	(*Valve 13, A+B*)
	(*spare*)
		Valve13FB
			(
			Enable_Motion:= Enable_Motion ,
			Enable_Latch:= TRUE,					(*Enabling Runs Valve as detent type (maintained solenoids*)
			Enable_SideA_PreCharge:= FALSE,		(*Enabling Turns Side A PreCharge Active, reset when Side B is energized in Auto*)
			Enable_SideB_PreCharge:= FALSE,		(*Enabling Turns Side B PreCharge Active, reset when Side A is energized in Auto*)
			PreCharge_Time:= T#0.10S,
			Enable_Auto_Commands:= In_Auto,
			Enable_Manual_Commands:= In_Manual AND All_Robots_Clear,
			In_Manual_SideA_Command:= Discrete_In.ManReqs.24,
			In_Manual_SideB_Command:= Discrete_In.ManReqs.25,
			SideA_Indicator:= FALSE,
			SideB_Indicator:= FALSE,
			TurnOn_SideA_SOL=> N100.Q.24,
			TurnOn_SideB_SOL=> N100.Q.25,
			TurnOn_SideA_Indicator=> Manual_Indicators1.24,
			TurnOn_SideB_Indicator=> Manual_Indicators1.25
			 );
		Valve13FB.In_Auto_SideA_Command:= FALSE;
		Valve13FB.In_Auto_SideB_Command:= FALSE;


	(*Valve 14, A+B*)
	(*spare*)
		Valve14FB
			(
			Enable_Motion:= Enable_Motion ,
			Enable_Latch:= TRUE,					(*Enabling Runs Valve as detent type (maintained solenoids*)
			Enable_SideA_PreCharge:= FALSE,		(*Enabling Turns Side A PreCharge Active, reset when Side B is energized in Auto*)
			Enable_SideB_PreCharge:= FALSE,		(*Enabling Turns Side B PreCharge Active, reset when Side A is energized in Auto*)
			PreCharge_Time:= T#0.10S,
			Enable_Auto_Commands:= In_Auto,
			Enable_Manual_Commands:= In_Manual AND All_Robots_Clear,
			In_Manual_SideA_Command:= Discrete_In.ManReqs.26,
			In_Manual_SideB_Command:= Discrete_In.ManReqs.27,
			SideA_Indicator:= FALSE,
			SideB_Indicator:= FALSE,
			TurnOn_SideA_SOL=> N100.Q.26,
			TurnOn_SideB_SOL=> N100.Q.27,
			TurnOn_SideA_Indicator=> Manual_Indicators1.26,
			TurnOn_SideB_Indicator=> Manual_Indicators1.27
			 );
		Valve14FB.In_Auto_SideA_Command:= FALSE;
		Valve14FB.In_Auto_SideB_Command:= FALSE;


	(*Valve 15, A+B*)
	(*spare*)
		Valve15FB
			(
			Enable_Motion:= Enable_Motion ,
			Enable_Latch:= TRUE,					(*Enabling Runs Valve as detent type (maintained solenoids*)
			Enable_SideA_PreCharge:= FALSE,		(*Enabling Turns Side A PreCharge Active, reset when Side B is energized in Auto*)
			Enable_SideB_PreCharge:= FALSE,		(*Enabling Turns Side B PreCharge Active, reset when Side A is energized in Auto*)
			PreCharge_Time:= T#0.10S,
			Enable_Auto_Commands:= In_Auto,
			Enable_Manual_Commands:= In_Manual AND All_Robots_Clear,
			In_Manual_SideA_Command:= Discrete_In.ManReqs.28,
			In_Manual_SideB_Command:= Discrete_In.ManReqs.29,
			SideA_Indicator:= FALSE,
			SideB_Indicator:= FALSE,
			TurnOn_SideA_SOL=> N100.Q.28,
			TurnOn_SideB_SOL=> N100.Q.29,
			TurnOn_SideA_Indicator=> Manual_Indicators1.28,
			TurnOn_SideB_Indicator=> Manual_Indicators1.29
			 );
		Valve15FB.In_Auto_SideA_Command:= FALSE;
		Valve15FB.In_Auto_SideB_Command:= FALSE;


	(*Valve 16, A+B*)
	(*spare*)
		Valve16FB
			(
			Enable_Motion:= Enable_Motion ,
			Enable_Latch:= TRUE,					(*Enabling Runs Valve as detent type (maintained solenoids*)
			Enable_SideA_PreCharge:= FALSE,		(*Enabling Turns Side A PreCharge Active, reset when Side B is energized in Auto*)
			Enable_SideB_PreCharge:= FALSE,		(*Enabling Turns Side B PreCharge Active, reset when Side A is energized in Auto*)
			PreCharge_Time:= T#0.10S,
			Enable_Auto_Commands:= In_Auto,
			Enable_Manual_Commands:= In_Manual AND All_Robots_Clear,
			In_Manual_SideA_Command:= Discrete_In.ManReqs.30,
			In_Manual_SideB_Command:= Discrete_In.ManReqs.31,
			SideA_Indicator:= FALSE,
			SideB_Indicator:= FALSE,
			TurnOn_SideA_SOL=> N100.Q.30,
			TurnOn_SideB_SOL=> N100.Q.31,
			TurnOn_SideA_Indicator=> Manual_Indicators1.30,
			TurnOn_SideB_Indicator=> Manual_Indicators1.31
			 );
		Valve16FB.In_Auto_SideA_Command:= FALSE;
		Valve16FB.In_Auto_SideB_Command:= FALSE;


























(*end*)
END_ACTION

ACTION ValveBank2:


(*+++++++++++THIS AREA IS CUSTOM PER INSTALLATION AND WILL HAVE TO BE MODIFIED PER +++++++++++++*)
(*+++++++++++THIS AREA IS CUSTOM PER INSTALLATION AND WILL HAVE TO BE MODIFIED PER +++++++++++++*)
(*+++++++++++THIS AREA IS CUSTOM PER INSTALLATION AND WILL HAVE TO BE MODIFIED PER +++++++++++++*)

(*+++++++++++VALVE BANK 2 +++++++++++++*)
(*+++++++++++VALVE BANK 2 +++++++++++++*)
(*+++++++++++VALVE BANK 2 +++++++++++++*)


	(*Valve 17, A+B*)
	(*spare*)
		Valve17FB
			(
			Enable_Motion:= Enable_Motion ,
			Enable_Latch:= TRUE,					(*Enabling Runs Valve as detent type (maintained solenoids*)
			Enable_SideA_PreCharge:= FALSE,		(*Enabling Turns Side A PreCharge Active, reset when Side B is energized in Auto*)
			Enable_SideB_PreCharge:= FALSE,		(*Enabling Turns Side B PreCharge Active, reset when Side A is energized in Auto*)
			PreCharge_Time:= T#0.1S,
			Enable_Auto_Commands:= In_Auto,
			Enable_Manual_Commands:= In_Manual AND All_Robots_Clear,
			In_Manual_SideA_Command:= Discrete_In.ManReqs2.0,
			In_Manual_SideB_Command:= (Discrete_In.ManReqs2.1 OR Discrete_In.Go_Home),
			SideA_Indicator:= FALSE,
			SideB_Indicator:= FALSE,
			TurnOn_SideA_SOL=> N101.Q.0,
			TurnOn_SideB_SOL=> N101.Q.1,
			TurnOn_SideA_Indicator=> Manual_Indicators2.0,
			TurnOn_SideB_Indicator=> Manual_Indicators2.1
			 );
		Valve17FB.In_Auto_SideA_Command:= FALSE;
		Valve17FB.In_Auto_SideB_Command:= FALSE;


	(*Valve 18, A+B*)
	(*spare*)
		Valve18FB
			(
			Enable_Motion:= Enable_Motion ,
			Enable_Latch:= TRUE,					(*Enabling Runs Valve as detent type (maintained solenoids*)
			Enable_SideA_PreCharge:= FALSE,		(*Enabling Turns Side A PreCharge Active, reset when Side B is energized in Auto*)
			Enable_SideB_PreCharge:= FALSE,		(*Enabling Turns Side B PreCharge Active, reset when Side A is energized in Auto*)
			PreCharge_Time:= T#0.10S,
			Enable_Auto_Commands:= In_Auto,
			Enable_Manual_Commands:= In_Manual AND All_Robots_Clear,
			In_Manual_SideA_Command:= Discrete_In.ManReqs2.2,
			In_Manual_SideB_Command:= Discrete_In.ManReqs2.3,
			SideA_Indicator:= FALSE,
			SideB_Indicator:= FALSE,
			TurnOn_SideA_SOL=> N101.Q.2,
			TurnOn_SideB_SOL=> N101.Q.3,
			TurnOn_SideA_Indicator=> Manual_Indicators2.2,
			TurnOn_SideB_Indicator=> Manual_Indicators2.3
			 );
		Valve18FB.In_Auto_SideA_Command:= FALSE;
		Valve18FB.In_Auto_SideB_Command:= FALSE;

	(*Valve 19, A+B*)
	(*spare*)
		Valve19FB
			(
			Enable_Motion:= Enable_Motion ,
			Enable_Latch:= TRUE,					(*Enabling Runs Valve as detent type (maintained solenoids*)
			Enable_SideA_PreCharge:= FALSE,		(*Enabling Turns Side A PreCharge Active, reset when Side B is energized in Auto*)
			Enable_SideB_PreCharge:= FALSE,		(*Enabling Turns Side B PreCharge Active, reset when Side A is energized in Auto*)
			PreCharge_Time:= T#0.10S,
			Enable_Auto_Commands:= In_Auto,
			Enable_Manual_Commands:= In_Manual AND All_Robots_Clear,
			In_Manual_SideA_Command:= Discrete_In.ManReqs2.4,
			In_Manual_SideB_Command:= Discrete_In.ManReqs2.5,
			SideA_Indicator:= FALSE,
			SideB_Indicator:= FALSE,
			TurnOn_SideA_SOL=> N101.Q.4,
			TurnOn_SideB_SOL=> N101.Q.5,
			TurnOn_SideA_Indicator=> Manual_Indicators2.4,
			TurnOn_SideB_Indicator=> Manual_Indicators2.5
			 );
		Valve19FB.In_Auto_SideA_Command:= FALSE;
		Valve19FB.In_Auto_SideB_Command:= FALSE;


	(*Valve 20, A+B*)
	(*spare*)
		Valve20FB
			(
			Enable_Motion:= Enable_Motion ,
			Enable_Latch:= TRUE,					(*Enabling Runs Valve as detent type (maintained solenoids*)
			Enable_SideA_PreCharge:= FALSE,		(*Enabling Turns Side A PreCharge Active, reset when Side B is energized in Auto*)
			Enable_SideB_PreCharge:= FALSE,		(*Enabling Turns Side B PreCharge Active, reset when Side A is energized in Auto*)
			PreCharge_Time:= T#0.10S,
			Enable_Auto_Commands:= In_Auto,
			Enable_Manual_Commands:= In_Manual AND All_Robots_Clear,
			In_Manual_SideA_Command:= Discrete_In.ManReqs2.6,
			In_Manual_SideB_Command:= Discrete_In.ManReqs2.7,
			SideA_Indicator:= FALSE,
			SideB_Indicator:= FALSE,
			TurnOn_SideA_SOL=> N101.Q.6,
			TurnOn_SideB_SOL=> N101.Q.7,
			TurnOn_SideA_Indicator=> Manual_Indicators2.6,
			TurnOn_SideB_Indicator=> Manual_Indicators2.7
			 );
		Valve20FB.In_Auto_SideA_Command:= FALSE;
		Valve20FB.In_Auto_SideB_Command:= FALSE;


	(*Valve 21, A+B*)
	(*spare*)
		Valve21FB
			(
			Enable_Motion:= Enable_Motion ,
			Enable_Latch:= TRUE,					(*Enabling Runs Valve as detent type (maintained solenoids*)
			Enable_SideA_PreCharge:= FALSE,		(*Enabling Turns Side A PreCharge Active, reset when Side B is energized in Auto*)
			Enable_SideB_PreCharge:= FALSE,		(*Enabling Turns Side B PreCharge Active, reset when Side A is energized in Auto*)
			PreCharge_Time:= T#0.10S,
			Enable_Auto_Commands:= In_Auto,
			Enable_Manual_Commands:= In_Manual AND All_Robots_Clear,
			In_Manual_SideA_Command:= Discrete_In.ManReqs2.8,
			In_Manual_SideB_Command:= Discrete_In.ManReqs2.9,
			SideA_Indicator:= FALSE,
			SideB_Indicator:= FALSE,
			TurnOn_SideA_SOL=> N101.Q.8,
			TurnOn_SideB_SOL=> N101.Q.9,
			TurnOn_SideA_Indicator=> Manual_Indicators2.8,
			TurnOn_SideB_Indicator=> Manual_Indicators2.9
			 );
		Valve21FB.In_Auto_SideA_Command:= FALSE;
		Valve21FB.In_Auto_SideB_Command:= FALSE;


	(*Valve 22, A+B*)
	(*spare*)
		Valve22FB
			(
			Enable_Motion:= Enable_Motion ,
			Enable_Latch:= TRUE,					(*Enabling Runs Valve as detent type (maintained solenoids*)
			Enable_SideA_PreCharge:= FALSE,		(*Enabling Turns Side A PreCharge Active, reset when Side B is energized in Auto*)
			Enable_SideB_PreCharge:= FALSE,		(*Enabling Turns Side B PreCharge Active, reset when Side A is energized in Auto*)
			PreCharge_Time:= T#0.10S,
			Enable_Auto_Commands:= In_Auto,
			Enable_Manual_Commands:= In_Manual AND All_Robots_Clear,
			In_Manual_SideA_Command:= Discrete_In.ManReqs2.10,
			In_Manual_SideB_Command:= Discrete_In.ManReqs2.11,
			SideA_Indicator:= FALSE,
			SideB_Indicator:= FALSE,
			TurnOn_SideA_SOL=> N101.Q.10,
			TurnOn_SideB_SOL=> N101.Q.11,
			TurnOn_SideA_Indicator=> Manual_Indicators2.10,
			TurnOn_SideB_Indicator=> Manual_Indicators2.11
			 );
		Valve22FB.In_Auto_SideA_Command:= FALSE;
		Valve22FB.In_Auto_SideB_Command:= FALSE;


	(*Valve 23, A+B*)
	(*spare*)
		Valve23FB
			(
			Enable_Motion:= Enable_Motion ,
			Enable_Latch:= TRUE,					(*Enabling Runs Valve as detent type (maintained solenoids*)
			Enable_SideA_PreCharge:= FALSE,		(*Enabling Turns Side A PreCharge Active, reset when Side B is energized in Auto*)
			Enable_SideB_PreCharge:= FALSE,		(*Enabling Turns Side B PreCharge Active, reset when Side A is energized in Auto*)
			PreCharge_Time:= T#0.10S,
			Enable_Auto_Commands:= In_Auto,
			Enable_Manual_Commands:= In_Manual AND All_Robots_Clear,
			In_Manual_SideA_Command:= Discrete_In.ManReqs2.12,
			In_Manual_SideB_Command:= Discrete_In.ManReqs2.13,
			SideA_Indicator:= FALSE,
			SideB_Indicator:= FALSE,
			TurnOn_SideA_SOL=> N101.Q.12,
			TurnOn_SideB_SOL=> N101.Q.13,
			TurnOn_SideA_Indicator=> Manual_Indicators2.12,
			TurnOn_SideB_Indicator=> Manual_Indicators2.13
			 );
		Valve23FB.In_Auto_SideA_Command:= FALSE;
		Valve23FB.In_Auto_SideB_Command:= FALSE;


	(*Valve 24, A+B*)
	(*spare*)
		Valve24FB
			(
			Enable_Motion:= Enable_Motion ,
			Enable_Latch:= TRUE,					(*Enabling Runs Valve as detent type (maintained solenoids*)
			Enable_SideA_PreCharge:= FALSE,		(*Enabling Turns Side A PreCharge Active, reset when Side B is energized in Auto*)
			Enable_SideB_PreCharge:= FALSE,		(*Enabling Turns Side B PreCharge Active, reset when Side A is energized in Auto*)
			PreCharge_Time:= T#0.10S,
			Enable_Auto_Commands:= In_Auto,
			Enable_Manual_Commands:= In_Manual AND All_Robots_Clear,
			In_Manual_SideA_Command:= Discrete_In.ManReqs2.14,
			In_Manual_SideB_Command:= Discrete_In.ManReqs2.15,
			SideA_Indicator:= FALSE,
			SideB_Indicator:= FALSE,
			TurnOn_SideA_SOL=> N101.Q.14,
			TurnOn_SideB_SOL=> N101.Q.15,
			TurnOn_SideA_Indicator=> Manual_Indicators2.14,
			TurnOn_SideB_Indicator=> Manual_Indicators2.15
			 );
		Valve24FB.In_Auto_SideA_Command:= FALSE;
		Valve24FB.In_Auto_SideB_Command:= FALSE;


	(*Valve 25, A+B*)
	(*spare*)
		Valve25FB
			(
			Enable_Motion:= Enable_Motion ,
			Enable_Latch:= TRUE,					(*Enabling Runs Valve as detent type (maintained solenoids*)
			Enable_SideA_PreCharge:= FALSE,		(*Enabling Turns Side A PreCharge Active, reset when Side B is energized in Auto*)
			Enable_SideB_PreCharge:= FALSE,		(*Enabling Turns Side B PreCharge Active, reset when Side A is energized in Auto*)
			PreCharge_Time:= T#0.10S,
			Enable_Auto_Commands:= In_Auto,
			Enable_Manual_Commands:= In_Manual AND All_Robots_Clear,
			In_Manual_SideA_Command:= Discrete_In.ManReqs2.16,
			In_Manual_SideB_Command:= Discrete_In.ManReqs2.17,
			SideA_Indicator:= FALSE,
			SideB_Indicator:= FALSE,
			TurnOn_SideA_SOL=> N101.Q.16,
			TurnOn_SideB_SOL=> N101.Q.17,
			TurnOn_SideA_Indicator=> Manual_Indicators2.16,
			TurnOn_SideB_Indicator=> Manual_Indicators2.17
			 );
		Valve25FB.In_Auto_SideA_Command:= FALSE;
		Valve25FB.In_Auto_SideB_Command:= FALSE;


	(*Valve 26, A+B*)
	(*spare*)
		Valve26FB
			(
			Enable_Motion:= Enable_Motion ,
			Enable_Latch:= TRUE,					(*Enabling Runs Valve as detent type (maintained solenoids*)
			Enable_SideA_PreCharge:= FALSE,		(*Enabling Turns Side A PreCharge Active, reset when Side B is energized in Auto*)
			Enable_SideB_PreCharge:= FALSE,		(*Enabling Turns Side B PreCharge Active, reset when Side A is energized in Auto*)
			PreCharge_Time:= T#0.10S,
			Enable_Auto_Commands:= In_Auto,
			Enable_Manual_Commands:= In_Manual AND All_Robots_Clear,
			In_Manual_SideA_Command:= Discrete_In.ManReqs2.18,
			In_Manual_SideB_Command:= Discrete_In.ManReqs2.19,
			SideA_Indicator:= FALSE,
			SideB_Indicator:= FALSE,
			TurnOn_SideA_SOL=> N101.Q.18,
			TurnOn_SideB_SOL=> N101.Q.19,
			TurnOn_SideA_Indicator=> Manual_Indicators2.18,
			TurnOn_SideB_Indicator=> Manual_Indicators2.19
			 );
		Valve26FB.In_Auto_SideA_Command:= FALSE;
		Valve26FB.In_Auto_SideB_Command:= FALSE;


	(*Valve 27, A+B*)
	(*spare*)
		Valve27FB
			(
			Enable_Motion:= Enable_Motion ,
			Enable_Latch:= TRUE,					(*Enabling Runs Valve as detent type (maintained solenoids*)
			Enable_SideA_PreCharge:= FALSE,		(*Enabling Turns Side A PreCharge Active, reset when Side B is energized in Auto*)
			Enable_SideB_PreCharge:= FALSE,		(*Enabling Turns Side B PreCharge Active, reset when Side A is energized in Auto*)
			PreCharge_Time:= T#0.10S,
			Enable_Auto_Commands:= In_Auto,
			Enable_Manual_Commands:= In_Manual AND All_Robots_Clear,
			In_Manual_SideA_Command:= Discrete_In.ManReqs2.20,
			In_Manual_SideB_Command:= Discrete_In.ManReqs2.21,
			SideA_Indicator:= FALSE,
			SideB_Indicator:= FALSE,
			TurnOn_SideA_SOL=> N101.Q.20,
			TurnOn_SideB_SOL=> N101.Q.21,
			TurnOn_SideA_Indicator=> Manual_Indicators2.20,
			TurnOn_SideB_Indicator=> Manual_Indicators2.21
			 );
		Valve27FB.In_Auto_SideA_Command:= FALSE;
		Valve27FB.In_Auto_SideB_Command:= FALSE;


	(*Valve 28, A+B*)
	(*spare*)
		Valve28FB
			(
			Enable_Motion:= Enable_Motion ,
			Enable_Latch:= TRUE,					(*Enabling Runs Valve as detent type (maintained solenoids*)
			Enable_SideA_PreCharge:= FALSE,		(*Enabling Turns Side A PreCharge Active, reset when Side B is energized in Auto*)
			Enable_SideB_PreCharge:= FALSE,		(*Enabling Turns Side B PreCharge Active, reset when Side A is energized in Auto*)
			PreCharge_Time:= T#0.10S,
			Enable_Auto_Commands:= In_Auto,
			Enable_Manual_Commands:= In_Manual AND All_Robots_Clear,
			In_Manual_SideA_Command:= Discrete_In.ManReqs2.22,
			In_Manual_SideB_Command:= Discrete_In.ManReqs2.23,
			SideA_Indicator:= FALSE,
			SideB_Indicator:= FALSE,
			TurnOn_SideA_SOL=> N101.Q.22,
			TurnOn_SideB_SOL=> N101.Q.23,
			TurnOn_SideA_Indicator=> Manual_Indicators2.22,
			TurnOn_SideB_Indicator=> Manual_Indicators2.23
			 );
		Valve28FB.In_Auto_SideA_Command:= FALSE;
		Valve28FB.In_Auto_SideB_Command:= FALSE;


	(*Valve 29, A+B*)
	(*spare*)
		Valve29FB
			(
			Enable_Motion:= Enable_Motion ,
			Enable_Latch:= TRUE,					(*Enabling Runs Valve as detent type (maintained solenoids*)
			Enable_SideA_PreCharge:= FALSE,		(*Enabling Turns Side A PreCharge Active, reset when Side B is energized in Auto*)
			Enable_SideB_PreCharge:= FALSE,		(*Enabling Turns Side B PreCharge Active, reset when Side A is energized in Auto*)
			PreCharge_Time:= T#0.10S,
			Enable_Auto_Commands:= In_Auto,
			Enable_Manual_Commands:= In_Manual AND All_Robots_Clear,
			In_Manual_SideA_Command:= Discrete_In.ManReqs2.24,
			In_Manual_SideB_Command:= Discrete_In.ManReqs2.25,
			SideA_Indicator:= FALSE,
			SideB_Indicator:= FALSE,
			TurnOn_SideA_SOL=> N101.Q.24,
			TurnOn_SideB_SOL=> N101.Q.25,
			TurnOn_SideA_Indicator=> Manual_Indicators2.24,
			TurnOn_SideB_Indicator=> Manual_Indicators2.25
			 );
		Valve29FB.In_Auto_SideA_Command:= FALSE;
		Valve29FB.In_Auto_SideB_Command:= FALSE;


	(*Valve 30, A+B*)
	(*spare*)
		Valve30FB
			(
			Enable_Motion:= Enable_Motion ,
			Enable_Latch:= TRUE,					(*Enabling Runs Valve as detent type (maintained solenoids*)
			Enable_SideA_PreCharge:= FALSE,		(*Enabling Turns Side A PreCharge Active, reset when Side B is energized in Auto*)
			Enable_SideB_PreCharge:= FALSE,		(*Enabling Turns Side B PreCharge Active, reset when Side A is energized in Auto*)
			PreCharge_Time:= T#0.10S,
			Enable_Auto_Commands:= In_Auto,
			Enable_Manual_Commands:= In_Manual AND All_Robots_Clear,
			In_Manual_SideA_Command:= Discrete_In.ManReqs2.26,
			In_Manual_SideB_Command:= Discrete_In.ManReqs2.27,
			SideA_Indicator:= FALSE,
			SideB_Indicator:= FALSE,
			TurnOn_SideA_SOL=> N101.Q.26,
			TurnOn_SideB_SOL=> N101.Q.27,
			TurnOn_SideA_Indicator=> Manual_Indicators2.26,
			TurnOn_SideB_Indicator=> Manual_Indicators2.27
			 );
		Valve30FB.In_Auto_SideA_Command:= FALSE;
		Valve30FB.In_Auto_SideB_Command:= FALSE;


	(*Valve 31, A+B*)
	(*spare*)
		Valve31FB
			(
			Enable_Motion:= Enable_Motion ,
			Enable_Latch:= TRUE,					(*Enabling Runs Valve as detent type (maintained solenoids*)
			Enable_SideA_PreCharge:= FALSE,		(*Enabling Turns Side A PreCharge Active, reset when Side B is energized in Auto*)
			Enable_SideB_PreCharge:= FALSE,		(*Enabling Turns Side B PreCharge Active, reset when Side A is energized in Auto*)
			PreCharge_Time:= T#0.10S,
			Enable_Auto_Commands:= In_Auto,
			Enable_Manual_Commands:= In_Manual AND All_Robots_Clear,
			In_Manual_SideA_Command:= Discrete_In.ManReqs2.28,
			In_Manual_SideB_Command:= Discrete_In.ManReqs2.29,
			SideA_Indicator:= FALSE,
			SideB_Indicator:= FALSE,
			TurnOn_SideA_SOL=> N101.Q.28,
			TurnOn_SideB_SOL=> N101.Q.29,
			TurnOn_SideA_Indicator=> Manual_Indicators2.28,
			TurnOn_SideB_Indicator=> Manual_Indicators2.29
			 );
		Valve31FB.In_Auto_SideA_Command:= FALSE;
		Valve31FB.In_Auto_SideB_Command:= FALSE;


	(*Valve 32, A+B*)
	(*spare*)
		Valve32FB
			(
			Enable_Motion:= Enable_Motion ,
			Enable_Latch:= TRUE,					(*Enabling Runs Valve as detent type (maintained solenoids*)
			Enable_SideA_PreCharge:= FALSE,		(*Enabling Turns Side A PreCharge Active, reset when Side B is energized in Auto*)
			Enable_SideB_PreCharge:= FALSE,		(*Enabling Turns Side B PreCharge Active, reset when Side A is energized in Auto*)
			PreCharge_Time:= T#0.10S,
			Enable_Auto_Commands:= In_Auto,
			Enable_Manual_Commands:= In_Manual AND All_Robots_Clear,
			In_Manual_SideA_Command:= Discrete_In.ManReqs2.30,
			In_Manual_SideB_Command:= Discrete_In.ManReqs2.31,
			SideA_Indicator:= FALSE,
			SideB_Indicator:= FALSE,
			TurnOn_SideA_SOL=> N101.Q.30,
			TurnOn_SideB_SOL=> N101.Q.31,
			TurnOn_SideA_Indicator=> Manual_Indicators2.30,
			TurnOn_SideB_Indicator=> Manual_Indicators2.31
			 );
		Valve32FB.In_Auto_SideA_Command:= FALSE;
		Valve32FB.In_Auto_SideB_Command:= FALSE;




















(*end*)
END_ACTION

ACTION ValveBank3:


(*+++++++++++THIS AREA IS CUSTOM PER INSTALLATION AND WILL HAVE TO BE MODIFIED PER +++++++++++++*)
(*+++++++++++THIS AREA IS CUSTOM PER INSTALLATION AND WILL HAVE TO BE MODIFIED PER +++++++++++++*)
(*+++++++++++THIS AREA IS CUSTOM PER INSTALLATION AND WILL HAVE TO BE MODIFIED PER +++++++++++++*)

(*+++++++++++VALVE BANK 3 +++++++++++++*)
(*+++++++++++VALVE BANK 3 +++++++++++++*)
(*+++++++++++VALVE BANK 3 +++++++++++++*)


	(*Valve 33, A+B*)
	(*spare*)
		Valve33FB
			(
			Enable_Motion:= Enable_Motion ,
			Enable_Latch:= TRUE,					(*Enabling Runs Valve as detent type (maintained solenoids*)
			Enable_SideA_PreCharge:= FALSE,		(*Enabling Turns Side A PreCharge Active, reset when Side B is energized in Auto*)
			Enable_SideB_PreCharge:= FALSE,		(*Enabling Turns Side B PreCharge Active, reset when Side A is energized in Auto*)
			PreCharge_Time:= T#0.1S,
			Enable_Auto_Commands:= In_Auto,
			Enable_Manual_Commands:= In_Manual AND All_Robots_Clear,
			In_Manual_SideA_Command:= Discrete_In.ManReqs3.0,
			In_Manual_SideB_Command:= (Discrete_In.ManReqs3.1 OR Discrete_In.Go_Home),
			SideA_Indicator:= FALSE,
			SideB_Indicator:= FALSE,
			TurnOn_SideA_SOL=> N102.Q.0,
			TurnOn_SideB_SOL=> N102.Q.1,
			TurnOn_SideA_Indicator=> Manual_Indicators3.0,
			TurnOn_SideB_Indicator=> Manual_Indicators3.1
			 );
		Valve33FB.In_Auto_SideA_Command:= FALSE;
		Valve33FB.In_Auto_SideB_Command:= FALSE;


	(*Valve 34, A+B*)
	(*spare*)
		Valve34FB
			(
			Enable_Motion:= Enable_Motion ,
			Enable_Latch:= TRUE,					(*Enabling Runs Valve as detent type (maintained solenoids*)
			Enable_SideA_PreCharge:= FALSE,		(*Enabling Turns Side A PreCharge Active, reset when Side B is energized in Auto*)
			Enable_SideB_PreCharge:= FALSE,		(*Enabling Turns Side B PreCharge Active, reset when Side A is energized in Auto*)
			PreCharge_Time:= T#0.10S,
			Enable_Auto_Commands:= In_Auto,
			Enable_Manual_Commands:= In_Manual AND All_Robots_Clear,
			In_Manual_SideA_Command:= Discrete_In.ManReqs3.2,
			In_Manual_SideB_Command:= Discrete_In.ManReqs3.3,
			SideA_Indicator:= FALSE,
			SideB_Indicator:= FALSE,
			TurnOn_SideA_SOL=> N102.Q.2,
			TurnOn_SideB_SOL=> N102.Q.3,
			TurnOn_SideA_Indicator=> Manual_Indicators3.2,
			TurnOn_SideB_Indicator=> Manual_Indicators3.3
			 );
		Valve34FB.In_Auto_SideA_Command:= FALSE;
		Valve34FB.In_Auto_SideB_Command:= FALSE;


	(*Valve 35, A+B*)
	(*spare*)
		Valve35FB
			(
			Enable_Motion:= Enable_Motion ,
			Enable_Latch:= TRUE,					(*Enabling Runs Valve as detent type (maintained solenoids*)
			Enable_SideA_PreCharge:= FALSE,		(*Enabling Turns Side A PreCharge Active, reset when Side B is energized in Auto*)
			Enable_SideB_PreCharge:= FALSE,		(*Enabling Turns Side B PreCharge Active, reset when Side A is energized in Auto*)
			PreCharge_Time:= T#0.10S,
			Enable_Auto_Commands:= In_Auto,
			Enable_Manual_Commands:= In_Manual AND All_Robots_Clear,
			In_Manual_SideA_Command:= Discrete_In.ManReqs3.4,
			In_Manual_SideB_Command:= Discrete_In.ManReqs3.5,
			SideA_Indicator:= FALSE,
			SideB_Indicator:= FALSE,
			TurnOn_SideA_SOL=> N102.Q.4,
			TurnOn_SideB_SOL=> N102.Q.5,
			TurnOn_SideA_Indicator=> Manual_Indicators3.4,
			TurnOn_SideB_Indicator=> Manual_Indicators3.5
			 );
		Valve35FB.In_Auto_SideA_Command:= FALSE;
		Valve35FB.In_Auto_SideB_Command:= FALSE;


	(*Valve 36, A+B*)
	(*spare*)
		Valve36FB
			(
			Enable_Motion:= Enable_Motion ,
			Enable_Latch:= TRUE,					(*Enabling Runs Valve as detent type (maintained solenoids*)
			Enable_SideA_PreCharge:= FALSE,		(*Enabling Turns Side A PreCharge Active, reset when Side B is energized in Auto*)
			Enable_SideB_PreCharge:= FALSE,		(*Enabling Turns Side B PreCharge Active, reset when Side A is energized in Auto*)
			PreCharge_Time:= T#0.10S,
			Enable_Auto_Commands:= In_Auto,
			Enable_Manual_Commands:= In_Manual AND All_Robots_Clear,
			In_Manual_SideA_Command:= Discrete_In.ManReqs3.6,
			In_Manual_SideB_Command:= Discrete_In.ManReqs3.7,
			SideA_Indicator:= FALSE,
			SideB_Indicator:= FALSE,
			TurnOn_SideA_SOL=> N102.Q.6,
			TurnOn_SideB_SOL=> N102.Q.7,
			TurnOn_SideA_Indicator=> Manual_Indicators3.6,
			TurnOn_SideB_Indicator=> Manual_Indicators3.7
			 );
		Valve36FB.In_Auto_SideA_Command:= FALSE;
		Valve36FB.In_Auto_SideB_Command:= FALSE;


	(*Valve 37, A+B*)
	(*spare*)
		Valve37FB
			(
			Enable_Motion:= Enable_Motion ,
			Enable_Latch:= TRUE,					(*Enabling Runs Valve as detent type (maintained solenoids*)
			Enable_SideA_PreCharge:= FALSE,		(*Enabling Turns Side A PreCharge Active, reset when Side B is energized in Auto*)
			Enable_SideB_PreCharge:= FALSE,		(*Enabling Turns Side B PreCharge Active, reset when Side A is energized in Auto*)
			PreCharge_Time:= T#0.10S,
			Enable_Auto_Commands:= In_Auto,
			Enable_Manual_Commands:= In_Manual AND All_Robots_Clear,
			In_Manual_SideA_Command:= Discrete_In.ManReqs3.8,
			In_Manual_SideB_Command:= Discrete_In.ManReqs3.9,
			SideA_Indicator:= FALSE,
			SideB_Indicator:= FALSE,
			TurnOn_SideA_SOL=> N102.Q.8,
			TurnOn_SideB_SOL=> N102.Q.9,
			TurnOn_SideA_Indicator=> Manual_Indicators3.8,
			TurnOn_SideB_Indicator=> Manual_Indicators3.9
			 );
		Valve37FB.In_Auto_SideA_Command:= FALSE;
		Valve37FB.In_Auto_SideB_Command:= FALSE;


	(*Valve 38, A+B*)
	(*spare*)
		Valve38FB
			(
			Enable_Motion:= Enable_Motion ,
			Enable_Latch:= TRUE,					(*Enabling Runs Valve as detent type (maintained solenoids*)
			Enable_SideA_PreCharge:= FALSE,		(*Enabling Turns Side A PreCharge Active, reset when Side B is energized in Auto*)
			Enable_SideB_PreCharge:= FALSE,		(*Enabling Turns Side B PreCharge Active, reset when Side A is energized in Auto*)
			PreCharge_Time:= T#0.10S,
			Enable_Auto_Commands:= In_Auto,
			Enable_Manual_Commands:= In_Manual AND All_Robots_Clear,
			In_Manual_SideA_Command:= Discrete_In.ManReqs3.10,
			In_Manual_SideB_Command:= Discrete_In.ManReqs3.11,
			SideA_Indicator:= FALSE,
			SideB_Indicator:= FALSE,
			TurnOn_SideA_SOL=> N102.Q.10,
			TurnOn_SideB_SOL=> N102.Q.11,
			TurnOn_SideA_Indicator=> Manual_Indicators3.10,
			TurnOn_SideB_Indicator=> Manual_Indicators3.11
			 );
		Valve38FB.In_Auto_SideA_Command:= FALSE;
		Valve38FB.In_Auto_SideB_Command:= FALSE;


	(*Valve 39, A+B*)
	(*spare*)
		Valve39FB
			(
			Enable_Motion:= Enable_Motion ,
			Enable_Latch:= TRUE,					(*Enabling Runs Valve as detent type (maintained solenoids*)
			Enable_SideA_PreCharge:= FALSE,		(*Enabling Turns Side A PreCharge Active, reset when Side B is energized in Auto*)
			Enable_SideB_PreCharge:= FALSE,		(*Enabling Turns Side B PreCharge Active, reset when Side A is energized in Auto*)
			PreCharge_Time:= T#0.10S,
			Enable_Auto_Commands:= In_Auto,
			Enable_Manual_Commands:= In_Manual AND All_Robots_Clear,
			In_Manual_SideA_Command:= Discrete_In.ManReqs3.12,
			In_Manual_SideB_Command:= Discrete_In.ManReqs3.13,
			SideA_Indicator:= FALSE,
			SideB_Indicator:= FALSE,
			TurnOn_SideA_SOL=> N102.Q.12,
			TurnOn_SideB_SOL=> N102.Q.13,
			TurnOn_SideA_Indicator=> Manual_Indicators3.12,
			TurnOn_SideB_Indicator=> Manual_Indicators3.13
			 );
		Valve39FB.In_Auto_SideA_Command:= FALSE;
		Valve39FB.In_Auto_SideB_Command:= FALSE;


	(*Valve 40, A+B*)
	(*spare*)
		Valve40FB
			(
			Enable_Motion:= Enable_Motion ,
			Enable_Latch:= TRUE,					(*Enabling Runs Valve as detent type (maintained solenoids*)
			Enable_SideA_PreCharge:= FALSE,		(*Enabling Turns Side A PreCharge Active, reset when Side B is energized in Auto*)
			Enable_SideB_PreCharge:= FALSE,		(*Enabling Turns Side B PreCharge Active, reset when Side A is energized in Auto*)
			PreCharge_Time:= T#0.10S,
			Enable_Auto_Commands:= In_Auto,
			Enable_Manual_Commands:= In_Manual AND All_Robots_Clear,
			In_Manual_SideA_Command:= Discrete_In.ManReqs3.14,
			In_Manual_SideB_Command:= Discrete_In.ManReqs3.15,
			SideA_Indicator:= FALSE,
			SideB_Indicator:= FALSE,
			TurnOn_SideA_SOL=> N102.Q.14,
			TurnOn_SideB_SOL=> N102.Q.15,
			TurnOn_SideA_Indicator=> Manual_Indicators3.14,
			TurnOn_SideB_Indicator=> Manual_Indicators3.15
			 );
		Valve40FB.In_Auto_SideA_Command:= FALSE;
		Valve40FB.In_Auto_SideB_Command:= FALSE;


	(*Valve 41, A+B*)
	(*spare*)
		Valve41FB
			(
			Enable_Motion:= Enable_Motion ,
			Enable_Latch:= TRUE,					(*Enabling Runs Valve as detent type (maintained solenoids*)
			Enable_SideA_PreCharge:= FALSE,		(*Enabling Turns Side A PreCharge Active, reset when Side B is energized in Auto*)
			Enable_SideB_PreCharge:= FALSE,		(*Enabling Turns Side B PreCharge Active, reset when Side A is energized in Auto*)
			PreCharge_Time:= T#0.10S,
			Enable_Auto_Commands:= In_Auto,
			Enable_Manual_Commands:= In_Manual AND All_Robots_Clear,
			In_Manual_SideA_Command:= Discrete_In.ManReqs3.16,
			In_Manual_SideB_Command:= Discrete_In.ManReqs3.17,
			SideA_Indicator:= FALSE,
			SideB_Indicator:= FALSE,
			TurnOn_SideA_SOL=> N102.Q.16,
			TurnOn_SideB_SOL=> N102.Q.17,
			TurnOn_SideA_Indicator=> Manual_Indicators3.16,
			TurnOn_SideB_Indicator=> Manual_Indicators3.17
			 );
		Valve41FB.In_Auto_SideA_Command:= FALSE;
		Valve41FB.In_Auto_SideB_Command:= FALSE;


	(*Valve 42, A+B*)
	(*spare*)
		Valve42FB
			(
			Enable_Motion:= Enable_Motion ,
			Enable_Latch:= TRUE,					(*Enabling Runs Valve as detent type (maintained solenoids*)
			Enable_SideA_PreCharge:= FALSE,		(*Enabling Turns Side A PreCharge Active, reset when Side B is energized in Auto*)
			Enable_SideB_PreCharge:= FALSE,		(*Enabling Turns Side B PreCharge Active, reset when Side A is energized in Auto*)
			PreCharge_Time:= T#0.10S,
			Enable_Auto_Commands:= In_Auto,
			Enable_Manual_Commands:= In_Manual AND All_Robots_Clear,
			In_Manual_SideA_Command:= Discrete_In.ManReqs3.18,
			In_Manual_SideB_Command:= Discrete_In.ManReqs3.19,
			SideA_Indicator:= FALSE,
			SideB_Indicator:= FALSE,
			TurnOn_SideA_SOL=> N102.Q.18,
			TurnOn_SideB_SOL=> N102.Q.19,
			TurnOn_SideA_Indicator=> Manual_Indicators3.18,
			TurnOn_SideB_Indicator=> Manual_Indicators3.19
			 );
		Valve42FB.In_Auto_SideA_Command:= FALSE;
		Valve42FB.In_Auto_SideB_Command:= FALSE;


	(*Valve 43, A+B*)
	(*spare*)
		Valve43FB
			(
			Enable_Motion:= Enable_Motion ,
			Enable_Latch:= TRUE,					(*Enabling Runs Valve as detent type (maintained solenoids*)
			Enable_SideA_PreCharge:= FALSE,		(*Enabling Turns Side A PreCharge Active, reset when Side B is energized in Auto*)
			Enable_SideB_PreCharge:= FALSE,		(*Enabling Turns Side B PreCharge Active, reset when Side A is energized in Auto*)
			PreCharge_Time:= T#0.10S,
			Enable_Auto_Commands:= In_Auto,
			Enable_Manual_Commands:= In_Manual AND All_Robots_Clear,
			In_Manual_SideA_Command:= Discrete_In.ManReqs3.20,
			In_Manual_SideB_Command:= Discrete_In.ManReqs3.21,
			SideA_Indicator:= FALSE,
			SideB_Indicator:= FALSE,
			TurnOn_SideA_SOL=> N102.Q.20,
			TurnOn_SideB_SOL=> N102.Q.21,
			TurnOn_SideA_Indicator=> Manual_Indicators3.20,
			TurnOn_SideB_Indicator=> Manual_Indicators3.21
			 );
		Valve43FB.In_Auto_SideA_Command:= FALSE;
		Valve43FB.In_Auto_SideB_Command:= FALSE;


	(*Valve 44, A+B*)
	(*spare*)
		Valve44FB
			(
			Enable_Motion:= Enable_Motion ,
			Enable_Latch:= TRUE,					(*Enabling Runs Valve as detent type (maintained solenoids*)
			Enable_SideA_PreCharge:= FALSE,		(*Enabling Turns Side A PreCharge Active, reset when Side B is energized in Auto*)
			Enable_SideB_PreCharge:= FALSE,		(*Enabling Turns Side B PreCharge Active, reset when Side A is energized in Auto*)
			PreCharge_Time:= T#0.10S,
			Enable_Auto_Commands:= In_Auto,
			Enable_Manual_Commands:= In_Manual AND All_Robots_Clear,
			In_Manual_SideA_Command:= Discrete_In.ManReqs3.22,
			In_Manual_SideB_Command:= Discrete_In.ManReqs3.23,
			SideA_Indicator:= FALSE,
			SideB_Indicator:= FALSE,
			TurnOn_SideA_SOL=> N102.Q.22,
			TurnOn_SideB_SOL=> N102.Q.23,
			TurnOn_SideA_Indicator=> Manual_Indicators3.22,
			TurnOn_SideB_Indicator=> Manual_Indicators3.23
			 );
		Valve44FB.In_Auto_SideA_Command:= FALSE;
		Valve44FB.In_Auto_SideB_Command:= FALSE;


	(*Valve 45, A+B*)
	(*spare*)
		Valve45FB
			(
			Enable_Motion:= Enable_Motion ,
			Enable_Latch:= TRUE,					(*Enabling Runs Valve as detent type (maintained solenoids*)
			Enable_SideA_PreCharge:= FALSE,		(*Enabling Turns Side A PreCharge Active, reset when Side B is energized in Auto*)
			Enable_SideB_PreCharge:= FALSE,		(*Enabling Turns Side B PreCharge Active, reset when Side A is energized in Auto*)
			PreCharge_Time:= T#0.10S,
			Enable_Auto_Commands:= In_Auto,
			Enable_Manual_Commands:= In_Manual AND All_Robots_Clear,
			In_Manual_SideA_Command:= Discrete_In.ManReqs3.24,
			In_Manual_SideB_Command:= Discrete_In.ManReqs3.25,
			SideA_Indicator:= FALSE,
			SideB_Indicator:= FALSE,
			TurnOn_SideA_SOL=> N102.Q.24,
			TurnOn_SideB_SOL=> N102.Q.25,
			TurnOn_SideA_Indicator=> Manual_Indicators3.24,
			TurnOn_SideB_Indicator=> Manual_Indicators3.25
			 );
		Valve45FB.In_Auto_SideA_Command:= FALSE;
		Valve45FB.In_Auto_SideB_Command:= FALSE;


	(*Valve 46, A+B*)
	(*spare*)
		Valve46FB
			(
			Enable_Motion:= Enable_Motion ,
			Enable_Latch:= TRUE,					(*Enabling Runs Valve as detent type (maintained solenoids*)
			Enable_SideA_PreCharge:= FALSE,		(*Enabling Turns Side A PreCharge Active, reset when Side B is energized in Auto*)
			Enable_SideB_PreCharge:= FALSE,		(*Enabling Turns Side B PreCharge Active, reset when Side A is energized in Auto*)
			PreCharge_Time:= T#0.10S,
			Enable_Auto_Commands:= In_Auto,
			Enable_Manual_Commands:= In_Manual AND All_Robots_Clear,
			In_Manual_SideA_Command:= Discrete_In.ManReqs3.26,
			In_Manual_SideB_Command:= Discrete_In.ManReqs3.27,
			SideA_Indicator:= FALSE,
			SideB_Indicator:= FALSE,
			TurnOn_SideA_SOL=> N102.Q.26,
			TurnOn_SideB_SOL=> N102.Q.27,
			TurnOn_SideA_Indicator=> Manual_Indicators3.26,
			TurnOn_SideB_Indicator=> Manual_Indicators3.27
			 );
		Valve46FB.In_Auto_SideA_Command:= FALSE;
		Valve46FB.In_Auto_SideB_Command:= FALSE;


	(*Valve 47, A+B*)
	(*spare*)
		Valve47FB
			(
			Enable_Motion:= Enable_Motion ,
			Enable_Latch:= TRUE,					(*Enabling Runs Valve as detent type (maintained solenoids*)
			Enable_SideA_PreCharge:= FALSE,		(*Enabling Turns Side A PreCharge Active, reset when Side B is energized in Auto*)
			Enable_SideB_PreCharge:= FALSE,		(*Enabling Turns Side B PreCharge Active, reset when Side A is energized in Auto*)
			PreCharge_Time:= T#0.10S,
			Enable_Auto_Commands:= In_Auto,
			Enable_Manual_Commands:= In_Manual AND All_Robots_Clear,
			In_Manual_SideA_Command:= Discrete_In.ManReqs3.28,
			In_Manual_SideB_Command:= Discrete_In.ManReqs3.29,
			SideA_Indicator:= FALSE,
			SideB_Indicator:= FALSE,
			TurnOn_SideA_SOL=> N102.Q.28,
			TurnOn_SideB_SOL=> N102.Q.29,
			TurnOn_SideA_Indicator=> Manual_Indicators3.28,
			TurnOn_SideB_Indicator=> Manual_Indicators3.29
			 );
		Valve47FB.In_Auto_SideA_Command:= FALSE;
		Valve47FB.In_Auto_SideB_Command:= FALSE;


	(*Valve 48, A+B*)
	(*spare*)
		Valve48FB
			(
			Enable_Motion:= Enable_Motion ,
			Enable_Latch:= TRUE,					(*Enabling Runs Valve as detent type (maintained solenoids*)
			Enable_SideA_PreCharge:= FALSE,		(*Enabling Turns Side A PreCharge Active, reset when Side B is energized in Auto*)
			Enable_SideB_PreCharge:= FALSE,		(*Enabling Turns Side B PreCharge Active, reset when Side A is energized in Auto*)
			PreCharge_Time:= T#0.10S,
			Enable_Auto_Commands:= In_Auto,
			Enable_Manual_Commands:= In_Manual AND All_Robots_Clear,
			In_Manual_SideA_Command:= Discrete_In.ManReqs3.30,
			In_Manual_SideB_Command:= Discrete_In.ManReqs3.31,
			SideA_Indicator:= FALSE,
			SideB_Indicator:= FALSE,
			TurnOn_SideA_SOL=> N102.Q.30,
			TurnOn_SideB_SOL=> N102.Q.31,
			TurnOn_SideA_Indicator=> Manual_Indicators3.30,
			TurnOn_SideB_Indicator=> Manual_Indicators3.31
			 );
		Valve48FB.In_Auto_SideA_Command:= FALSE;
		Valve48FB.In_Auto_SideB_Command:= FALSE;


























(*end*)
END_ACTION

ACTION Xfer_To_UI:
(*Transfer General Status of Fixture and I/O Images for Display On HMI*)
	Discrete_Image.Status:= Status;
	Discrete_Image.CLFaults1:= CLFaults1;
	Discrete_Image.CLFaults2:= CLFaults2;
	Discrete_Image.CLFaults3:= CLFaults3;
	Discrete_Image.CLFaults4:= CLFaults4;
	Discrete_Image.CLFaulted:= CLFaulted;
	Discrete_Image.PPFaults:= PPFaults;
	Discrete_Image.PPFaults1:= PPFaults1;
	Discrete_Image.PPFaults2:= PPFaults2;
	Discrete_Image.PPFaulted:= PPFaulted;
	Discrete_Image.Model_Data:= Model_ID;
	Discrete_Image.ToolID:= Fix_ID;
	Discrete_Image.ProdCount:= Prod_Count_Out;
	Discrete_Image.CycleTime:= Cycle_Time_Out;
	Discrete_Image.PrevCycleTime:= PrevCycle_Time_Out;
	Discrete_Image.LoadTime:= Load_Time_Out;
	Discrete_Image.WeldTime:= Weld_Time_Out;
	Discrete_Image.UnloadTime:= Unload_Time_Out;

	Discrete_Image.InAuto:= In_Auto_Mode;
	Discrete_Image.InManual:= In_Manual_Mode;
	Discrete_Image.ManInds:= Manual_Indicators1;
	Discrete_Image.ManInds2:= Manual_Indicators2;
	Discrete_Image.ManInds3:= Manual_Indicators3;
	Discrete_Image.At_Home:= Tool_At_Home;
	Discrete_Image.Enable_Motion:= Enable_Motion;
	Discrete_Image.All_Sensors_Off:= All_Sensors_Off;
	Discrete_Image.Bypass_ACKS:= Discrete_In.Bypass_REQS;
	Discrete_Image.CustomApplication_ACKS:= Discrete_In.CustomApplication_REQS;
	Discrete_Image.Fixture_Allow_Model_Change:= Fixture_Allow_Model_Change;
	Discrete_Image.NodeLayout:=NodeLayout;
	Discrete_Image.NodeState:=NodeState;
	
	Discrete_Image.Input_Node_Count:= Discrete_In.Input_Node_Count;
	Discrete_Image.VB_Node_Count:= Discrete_In.VB_Node_Count;
	Discrete_Image.Water_Stand_Count:= Discrete_In.Water_Stand_Count;

	IF  (Discrete_Image.Input_Node_Count < 4)
		THEN Discrete_Image.VB_Screen_Position:= 1;
	ELSIF  (Discrete_Image.Input_Node_Count < 7)
		THEN Discrete_Image.VB_Screen_Position:= 2;
	ELSIF  (Discrete_Image.Input_Node_Count < 10)
		THEN Discrete_Image.VB_Screen_Position:= 3;
	ELSIF  (Discrete_Image.Input_Node_Count < 13)
		THEN Discrete_Image.VB_Screen_Position:= 4;
	ELSIF  (Discrete_Image.Input_Node_Count < 16)
		THEN Discrete_Image.VB_Screen_Position:= 5;
	ELSIF  (Discrete_Image.Input_Node_Count < 19)
		THEN Discrete_Image.VB_Screen_Position:= 6;
	ELSIF  (Discrete_Image.Input_Node_Count < 22)
		THEN Discrete_Image.VB_Screen_Position:= 7;
	ELSIF  (Discrete_Image.Input_Node_Count < 26)
		THEN Discrete_Image.VB_Screen_Position:= 8;
	ELSE
			Discrete_Image.VB_Screen_Position:= 9;
	END_IF;

	Discrete_Image.N00:= N00;
	Discrete_Image.N01:= N01;
	Discrete_Image.N02:= N02;
	Discrete_Image.N03:= N03;
	Discrete_Image.N04:= N04;
	Discrete_Image.N05:= N05;
	Discrete_Image.N06:= N06;
	Discrete_Image.N07:= N07;
	Discrete_Image.N08:= N08;
	Discrete_Image.N09:= N09;
	Discrete_Image.N10:= N10;
	Discrete_Image.N11:= N11;
	Discrete_Image.N12:= N12;
	Discrete_Image.N13:= N13;
	Discrete_Image.N14:= N14;
	Discrete_Image.N15:= N15;
	Discrete_Image.N16:= N16;
	Discrete_Image.N17:= N17;
	Discrete_Image.N18:= N18;
	Discrete_Image.N19:= N19;
	Discrete_Image.N100:= N100;
	Discrete_Image.N100_STAT:= N100_STAT;
	Discrete_Image.N101:= N101;
	Discrete_Image.N101_STAT:= N101_STAT;
	Discrete_Image.N102:= N102;
	Discrete_Image.N102_STAT:= N102_STAT;


	Discrete_Image.ECatSlave_Cable_Breaks:= ECatSlave_Cable_Breaks;

	Discrete_Image.Operator_Performance_Pen:= Production_Report.Shift_Report[0].Prod_Performance;
END_ACTION

END_PROGRAM

// ---- POUs/Fixtures and EOAT/Not_Used/Fix11.TcPOU
(*Fixture*)

PROGRAM Fix11
	VAR_INPUT
		Enable_Prog: BOOL;
		Enable_Motion: BOOL;
		Discrete_In: udt_FixXX_Input_Image_20180202;
		Dry_Cycle: BOOL;
		Cell_In_Services: BOOL;
		Flash_Rate: BOOL;
		NodeLayout:udt_ECATNodeData_20221507;

	END_VAR

	VAR
(*Hardware Related Data Types*)
			(*Develop "Beckhoff Nodes"*)
			{attribute 'OPC.UA.DA':='1'}
			N00 AT %I*: udt_EP1111;
			{attribute 'OPC.UA.DA':='1'}
			N01 AT %I*: udt_EP1008_002_v2;
			{attribute 'OPC.UA.DA':='1'}
			N02 AT %I*: udt_EP1008_002_v2;
			{attribute 'OPC.UA.DA':='1'}
			N03 AT %I*: udt_EP1008_002_v2;
			{attribute 'OPC.UA.DA':='1'}
			N04 AT %I*: udt_EP1008_002_v2;
			{attribute 'OPC.UA.DA':='1'}
			N05 AT %I*: udt_EP1008_002_v2;
			{attribute 'OPC.UA.DA':='1'}
			N06 AT %I*: udt_EP1008_002_v2;
			{attribute 'OPC.UA.DA':='1'}
			N07 AT %I*: udt_EP1008_002_v2;
			{attribute 'OPC.UA.DA':='1'}
			N08 AT %I*: udt_EP1008_002_v2;
			{attribute 'OPC.UA.DA':='1'}
			N09 AT %I*: udt_EP1008_002_v2;
			{attribute 'OPC.UA.DA':='1'}
			N10 AT %I*: udt_EP1008_002_v2;
			{attribute 'OPC.UA.DA':='1'}
			N11 AT %I*: udt_EP1008_002_v2;
			{attribute 'OPC.UA.DA':='1'}
			N12 AT %I*: udt_EP1008_002_v2;
			{attribute 'OPC.UA.DA':='1'}
			N13 AT %I*: udt_EP1008_002_v2;
			{attribute 'OPC.UA.DA':='1'}
			N14 AT %I*: udt_EP1008_002_v2;
			{attribute 'OPC.UA.DA':='1'}
			N15 AT %I*: udt_EP1008_002_v2;
			{attribute 'OPC.UA.DA':='1'}
			N16 AT %I*: udt_EP1008_002_v2;
			{attribute 'OPC.UA.DA':='1'}
			N17 AT %I*: udt_EP1008_002_v2;
			{attribute 'OPC.UA.DA':='1'}
			N18 AT %I*: udt_EP1008_002_v2;
			{attribute 'OPC.UA.DA':='1'}
			N19 AT %I*: udt_EP1008_002_v2;
			{attribute 'OPC.UA.DA':='1'}
			N20 AT %I*: udt_EP1008_002_v2;
			{attribute 'OPC.UA.DA':='1'}
			N21 AT %I*: udt_EP1008_002_v2;
			{attribute 'OPC.UA.DA':='1'}
			N22 AT %I*: udt_EP1008_002_v2;
			{attribute 'OPC.UA.DA':='1'}
			N100 AT %Q*: udt_SMC_EX260_ValveBank;
			{attribute 'OPC.UA.DA':='1'}
			N100_STAT AT %I*:udt_SMC_EX260_Stat;
			{attribute 'OPC.UA.DA':='1'}
			N101 AT %Q*: udt_SMC_EX260_ValveBank;
			{attribute 'OPC.UA.DA':='1'}
			N101_STAT AT %I*:udt_SMC_EX260_Stat;
			{attribute 'OPC.UA.DA':='1'}
			N102 AT %Q*: udt_SMC_EX260_ValveBank;
			{attribute 'OPC.UA.DA':='1'}
			N102_STAT AT %I*:udt_SMC_EX260_Stat;

(* Nodes States*)
		NodeState: ARRAY[0..63] OF UINT;
		DiscreteNode_OK: BOOL;
(*Cable Break States*)
		ECatSlave_Cable_Breaks: ARRAY[0..1] OF DINT;
(*Standard Internal Variables*)
		(*Generic Sensor Variables*)
		All_Sensors_On: UINT;
		All_Sensors_Off: BOOL;
		All_Sensors_Off1: BOOL;
		All_Sensors_Off2: BOOL;
		(*Generic Position Variables*)
		Tool_At_Home: BOOL;
		Tool_At_Load: UINT;
		Tool_At_Weld: UINT;
		Tool_At_Rotate: UINT;
		Tool_At_Seal: UINT;
		Tool_At_Stud: UINT;
		Tool_At_Unload: UINT ;
		(*Grouping Of Items*)
		All_QAChecks_OK: BOOL;
		QAChecks_Failed: BOOL;
		(*General Internals*)
		In_Auto: BOOL;
		In_Manual: BOOL;

		Auto_Run: BOOL;
		Reset_All_Completes:BOOL;
		Load_Robots_Clear1: BOOL;
		Load_Robots_Clear2: BOOL;
		Load_Robots_Clear: BOOL;
		Load_Robots_WorkingOK1: BOOL;
		Load_Robots_WorkingOK2: BOOL;
		Load_Robots_Complete1: BOOL;
		Load_Robots_Complete2: BOOL;
		Load_Robots_PartInEOAT1: BOOL;
		Load_Robots_PartInEOAT2: BOOL;
		Load_Robots_UnclampEarly1: BOOL;
		Load_Robots_UnclampEarly2: BOOL;
		Seal_Robots_Clear: BOOL;
		Seal_Robots_WorkingOK: BOOL;
		Seal_Robots_UnclampEarly: BOOL;
		Seal_Robots_Complete: BOOL;
		Stud_Robots_Clear: BOOL;
		Stud_Robots_WorkingOK: BOOL;
		Stud_Robots_UnclampEarly: BOOL;
		Stud_Robots_Complete: BOOL;
		Weld_Robots_Clear: BOOL;
		Weld_Robots_WorkingOK: BOOL;
		Weld_Robots_UnclampEarly: BOOL;
		Weld_Robots_Complete: BOOL;
		Mig_Robots_Ready :BOOL;
		TurntableA_Clear: BOOL;
		TurntableB_Clear: BOOL;
		Turntable_Clear:BOOL;
		Turntable_WorkingOK: BOOL;
		TurntableA_Complete: BOOL;
		TurntableB_Complete: BOOL;
		Unload_Robots_Clear1: BOOL;
		Unload_Robots_WorkingOK1: BOOL;
		Unload_Robots_Complete1: BOOL;
		Unload_Robots_EOATEmpty1: BOOL;
		Unload_Robots_Clear2: BOOL;
		Unload_Robots_WorkingOK2: BOOL;
		Unload_Robots_Complete2: BOOL;
		Unload_Robots_EOATEmpty2: BOOL;
		Unload_Robots_Clear: BOOL;
		All_Robots_Clear: BOOL;

		Unload_Robot_Complete: BOOL;

		Start_Load_Robots1: BOOL;
		Start_Load_Robots2: BOOL;
		Start_Weld_Robots: BOOL;
		Start_Unload_Robots1: BOOL;
		Start_Unload_Robots2: BOOL;
		Start_Seal_Robots: BOOL;
		Start_Stud_Robots: BOOL;
		Start_TurntableA: BOOL;
		Start_TurntableB: BOOL;
		Load_Robots_Proceed1: BOOL;
		Load_Robots_Proceed2: BOOL;
		Weld_Robots_Proceed: BOOL;
		Seal_Robots_Proceed: BOOL;
		Stud_Robots_Proceed: BOOL;
		Unload_Robots_Proceed1: BOOL;
		Unload_Robots_Proceed2: BOOL;

		Prod_Inc: R_TRIG;
		Cycle_Time: TON;
		Cycle_Time_Pulse: R_TRIG;
		Load_Time: TON;
		Weld_Time: TON;
		Seal_Time: TON;
		Stud_Time: TON;
		Turn_Time: TON;
		Unload_Time: TON;
		Date_Stamp_TMR: TON;
		Date_StampHome_TMR: TON;
		CLFaulted: UDINT;
		PPFaulted: UDINT;
		Manual_Ind_HomePrompt: BOOL;
		Fixture_Allow_Model_Change: BOOL;

(*Non-Standard Variables*)

		(*FB Instances*)
		Clamp1FB: FB_Cylinder_Status;
		Clamp2FB: FB_Cylinder_Status;
		Clamp3FB: FB_Cylinder_Status;
		Clamp4FB: FB_Cylinder_Status;
		Clamp5FB: FB_Cylinder_Status;
		Clamp6FB: FB_Cylinder_Status;
		Clamp7FB: FB_Cylinder_Status;
		Clamp8FB: FB_Cylinder_Status;
		Clamp9FB: FB_Cylinder_Status;
		Clamp10FB: FB_Cylinder_Status;
		Clamp11FB: FB_Cylinder_Status;
		Clamp12FB: FB_Cylinder_Status;
		Clamp13FB: FB_Cylinder_Status;
		Clamp14FB: FB_Cylinder_Status;
		Clamp15FB: FB_Cylinder_Status;
		Clamp16FB: FB_Cylinder_Status;
		Clamp17FB: FB_Cylinder_Status;
		Clamp18FB: FB_Cylinder_Status;
		Clamp19FB: FB_Cylinder_Status;
		Clamp20FB: FB_Cylinder_Status;
		Clamp21FB: FB_Cylinder_Status;
		Clamp22FB: FB_Cylinder_Status;
		Clamp23FB: FB_Cylinder_Status;
		Clamp24FB: FB_Cylinder_Status;
		Cyl1FB: FB_TripleCylinder_20150625;
		Pin1FB: FB_Cylinder_Status;
		Pin2FB: FB_Cylinder_Status;
		Pin3FB: FB_Cylinder_Status;
		Pin4FB: FB_Cylinder_Status;
		Pin5FB: FB_Cylinder_Status;
		Pin6FB: FB_Cylinder_Status;
		Pin7FB: FB_Cylinder_Status;
		Pin8FB: FB_Cylinder_Status;
		Pin9FB: FB_Cylinder_Status;
		Pin10FB: FB_Cylinder_Status;
		Pin11FB: FB_Cylinder_Status;
		Pin12FB: FB_Cylinder_Status;
		Pin13FB: FB_Cylinder_Status;
		Pin14FB: FB_Cylinder_Status;
		Slide1FB: FB_Cylinder_Status;
		Slide2FB: FB_Cylinder_Status;
		Slide3FB: FB_Cylinder_Status;
		Slide4FB: FB_Cylinder_Status;
		Slide5FB: FB_Cylinder_Status;
		Slide6FB: FB_Cylinder_Status;
		Swing1FB: FB_Cylinder_Status;
		Swing2FB: FB_Cylinder_Status;
		Swing3FB: FB_Cylinder_Status;
		Swing4FB: FB_Cylinder_Status;
		Swing5FB: FB_Cylinder_Status;
		Swing6FB: FB_Cylinder_Status;
		QACheck1FB: FB_Cylinder_Status;
		QACheck2FB: FB_Cylinder_Status;
		CheckQA1FB: FB_GTAC_QAcheck_20150529;
		Part_Present1FB: FB_PP_Sensor;
		Part_Present2FB: FB_PP_Sensor;
		Part_Present3FB: FB_PP_Sensor;
		Part_Present4FB: FB_PP_Sensor;
		Part_Present5FB: FB_PP_Sensor;
		Part_Present6FB: FB_PP_Sensor;
		Part_Present7FB: FB_PP_Sensor;
		Part_Present8FB: FB_PP_Sensor;
		Part_Present9FB: FB_PP_Sensor;
		Part_Present10FB: FB_PP_Sensor;
		Part_Present11FB: FB_PP_Sensor;
		Part_Present12FB: FB_PP_Sensor;
		Part_Present13FB: FB_PP_Sensor;
		Part_Present14FB: FB_PP_Sensor;
		Part_Present15FB: FB_PP_Sensor;
		Part_Present16FB: FB_PP_Sensor;
		Part_Present17FB: FB_PP_Sensor;
		Part_Present18FB: FB_PP_Sensor;
		Part_Present19FB: FB_PP_Sensor;
		Part_Present20FB: FB_PP_Sensor;
		Part_Present21FB: FB_PP_Sensor;
		Part_Present22FB: FB_PP_Sensor;
		Part_Present23FB: FB_PP_Sensor;
		Part_Present24FB: FB_PP_Sensor;
		Part_Present25FB: FB_PP_Sensor;
		Part_Present26FB: FB_PP_Sensor;
		Part_Present27FB: FB_PP_Sensor;
		Part_Present28FB: FB_PP_Sensor;
		Part_Present29FB: FB_PP_Sensor;
		Part_Present30FB: FB_PP_Sensor;
		Part_Present31FB: FB_PP_Sensor;
		Part_Present32FB: FB_PP_Sensor;
		Part_Present33FB: FB_PP_Sensor;
		Part_Present34FB: FB_PP_Sensor;
		Part_Present35FB: FB_PP_Sensor;
		Part_Present36FB: FB_PP_Sensor;
		Part_Present37FB: FB_PP_Sensor;
		Part_Present38FB: FB_PP_Sensor;
		Part_Present39FB: FB_PP_Sensor;
		Part_Present40FB: FB_PP_Sensor;
		Tape_Present1FB: FB_PP_Sensor;

		(*Valve FBs*)
		Valve1FB: FB_GTAC_Valve_20170704;
		Valve2FB: FB_GTAC_Valve_20170704;
		Valve3FB: FB_GTAC_Valve_20170704;
		Valve4FB: FB_GTAC_Valve_20170704;
		Valve5FB: FB_GTAC_Valve_20170704;
		Valve6FB: FB_GTAC_Valve_20170704;
		Valve7FB: FB_GTAC_Valve_20170704;
		Valve8FB: FB_GTAC_Valve_20170704;
		Valve9FB: FB_GTAC_Valve_20170704;
		Valve10FB: FB_GTAC_Valve_20170704;
		Valve11FB: FB_GTAC_Valve_20170704;
		Valve12FB: FB_GTAC_Valve_20170704;
		Valve13FB: FB_GTAC_Valve_20170704;
		Valve14FB: FB_GTAC_Valve_20170704;
		Valve15FB: FB_GTAC_Valve_20170704;
		Valve16FB: FB_GTAC_Valve_20170704;
		Valve17FB: FB_GTAC_Valve_20170704;
		Valve18FB: FB_GTAC_Valve_20170704;
		Valve19FB: FB_GTAC_Valve_20170704;
		Valve20FB: FB_GTAC_Valve_20170704;
		Valve21FB: FB_GTAC_Valve_20170704;
		Valve22FB: FB_GTAC_Valve_20170704;
		Valve23FB: FB_GTAC_Valve_20170704;
		Valve24FB: FB_GTAC_Valve_20170704;
		Valve25FB: FB_GTAC_Valve_20170704;
		Valve26FB: FB_GTAC_Valve_20170704;
		Valve27FB: FB_GTAC_Valve_20170704;
		Valve28FB: FB_GTAC_Valve_20170704;
		Valve29FB: FB_GTAC_Valve_20170704;
		Valve30FB: FB_GTAC_Valve_20170704;
		Valve31FB: FB_GTAC_Valve_20170704;
		Valve32FB: FB_GTAC_Valve_20170704;
		Valve33FB: FB_GTAC_Valve_20170704;
		Valve34FB: FB_GTAC_Valve_20170704;
		Valve35FB: FB_GTAC_Valve_20170704;
		Valve36FB: FB_GTAC_Valve_20170704;
		Valve37FB: FB_GTAC_Valve_20170704;
		Valve38FB: FB_GTAC_Valve_20170704;
		Valve39FB: FB_GTAC_Valve_20170704;
		Valve40FB: FB_GTAC_Valve_20170704;
		Valve41FB: FB_GTAC_Valve_20170704;
		Valve42FB: FB_GTAC_Valve_20170704;
		Valve43FB: FB_GTAC_Valve_20170704;
		Valve44FB: FB_GTAC_Valve_20170704;
		Valve45FB: FB_GTAC_Valve_20170704;
		Valve46FB: FB_GTAC_Valve_20170704;
		Valve47FB: FB_GTAC_Valve_20170704;
		Valve48FB: FB_GTAC_Valve_20170704;

		(*Tool Positions*)
			(*Add User Indivdual Position Variables Here*)
			Clamp1ADVD: BOOL;
			Clamp1RETD: BOOL;
			Clamp2ADVD: BOOL;
			Clamp2RETD: BOOL;
			Clamp3ADVD: BOOL;
			Clamp3RETD: BOOL;
			Clamp4ADVD: BOOL;
			Clamp4RETD: BOOL;
			Clamp5ADVD: BOOL;
			Clamp5RETD: BOOL;
			Clamp6ADVD: BOOL;
			Clamp6RETD: BOOL;
			Clamp7ADVD: BOOL;
			Clamp7RETD: BOOL;
			Clamp8ADVD: BOOL;
			Clamp8RETD: BOOL;
			Clamp9ADVD: BOOL;
			Clamp9RETD: BOOL;
			Clamp10ADVD: BOOL;
			Clamp10RETD: BOOL;
			Clamp11ADVD: BOOL;
			Clamp11RETD: BOOL;
			Clamp12ADVD: BOOL;
			Clamp12RETD: BOOL;
			Clamp13ADVD: BOOL;
			Clamp13RETD: BOOL;
			Clamp14ADVD: BOOL;
			Clamp14RETD: BOOL;
			Clamp15ADVD: BOOL;
			Clamp15RETD: BOOL;
			Clamp16ADVD: BOOL;
			Clamp16RETD: BOOL;
			Clamp17ADVD: BOOL;
			Clamp17RETD: BOOL;
			Clamp18ADVD: BOOL;
			Clamp18RETD: BOOL;
			Clamp19ADVD: BOOL;
			Clamp19RETD: BOOL;
			Clamp20ADVD: BOOL;
			Clamp20RETD: BOOL;
			Clamp21ADVD: BOOL;
			Clamp21RETD: BOOL;
			Clamp22ADVD: BOOL;
			Clamp22RETD: BOOL;
			Clamp23ADVD: BOOL;
			Clamp23RETD: BOOL;
			Clamp24ADVD: BOOL;
			Clamp24RETD: BOOL;
			Cyl1ADVD: BOOL;
			Cyl1MID: BOOL;
			Cyl1RETD: BOOL;
			Pin1ADVD: BOOL;
			Pin1RETD: BOOL;
			Pin2ADVD: BOOL;
			Pin2RETD: BOOL;
			Pin3ADVD: BOOL;
			Pin3RETD: BOOL;
			Pin4ADVD: BOOL;
			Pin4RETD: BOOL;
			Pin5ADVD: BOOL;
			Pin5RETD: BOOL;
			Pin6ADVD: BOOL;
			Pin6RETD: BOOL;
			Pin7ADVD: BOOL;
			Pin7RETD: BOOL;
			Pin8ADVD: BOOL;
			Pin8RETD: BOOL;
			Pin9ADVD: BOOL;
			Pin9RETD: BOOL;
			Pin10ADVD: BOOL;
			Pin10RETD: BOOL;
			Pin11ADVD: BOOL;
			Pin11RETD: BOOL;
			Pin12ADVD: BOOL;
			Pin12RETD: BOOL;
			Pin13ADVD: BOOL;
			Pin13RETD: BOOL;
			Pin14ADVD: BOOL;
			Pin14RETD: BOOL;
			Slide1ADVD: BOOL;
			Slide1RETD: BOOL;
			Slide2ADVD: BOOL;
			Slide2RETD: BOOL;
			Slide3ADVD: BOOL;
			Slide3RETD: BOOL;
			Slide4ADVD: BOOL;
			Slide4RETD: BOOL;
			Slide5ADVD: BOOL;
			Slide5RETD: BOOL;
			Slide6ADVD: BOOL;
			Slide6RETD: BOOL;
			Swing1ADVD: BOOL;
			Swing1RETD: BOOL;
			Swing2ADVD: BOOL;
			Swing2RETD: BOOL;
			Swing3ADVD: BOOL;
			Swing3RETD: BOOL;
			Swing4ADVD: BOOL;
			Swing4RETD: BOOL;
			Swing5ADVD: BOOL;
			Swing5RETD: BOOL;
			Swing6ADVD: BOOL;
			Swing6RETD: BOOL;
			QACheck1ADVD: BOOL;
			QACheck1RETD: BOOL;
			QACheck2ADVD: BOOL;
			QACheck2RETD: BOOL;

		(*Part Present Sensors*)
			(*Main Body Present*)
			Part_Present1: BOOL;
			Part_Present2: BOOL;
			Part_Present3: BOOL;
			Part_Present4: BOOL;
			Part_Present5: BOOL;
			Part_Present6: BOOL;
			Part_Present7: BOOL;
			Part_Present8: BOOL;
			Part_Present9: BOOL;
			Part_Present10: BOOL;
			Part_Present11: BOOL;
			Part_Present12: BOOL;
			Part_Present13: BOOL;
			Part_Present14: BOOL;
			Part_Present15: BOOL;
			Part_Present16: BOOL;
			Part_Present17: BOOL;
			Part_Present18: BOOL;
			Part_Present19: BOOL;
			Part_Present20: BOOL;
			Part_Present21: BOOL;
			Part_Present22: BOOL;
			Part_Present23: BOOL;
			Part_Present24: BOOL;
			Part_Present25: BOOL;
			Part_Present26: BOOL;
			Part_Present27: BOOL;
			Part_Present28: BOOL;
			Part_Present29: BOOL;
			Part_Present30: BOOL;
			Part_Present31: BOOL;
			Part_Present32: BOOL;
			Part_Present33: BOOL;
			Part_Present34: BOOL;
			Part_Present35: BOOL;
			Part_Present36: BOOL;
			Part_Present37: BOOL;
			Part_Present38: BOOL;
			Part_Present39: BOOL;
			Part_Present40: BOOL;
			Tape_Present1: BOOL;

		(*Motion Sequence Variables*)
			Clamp_Step: UINT;
			Repo1_Step: UINT;
			Repo2_Step: UINT;
			Repo3_Step: UINT;
			Repo4_Step: UINT;
			Unclamp_Step: UINT;

		(*Custom Application Variables*)
			Weld_Curtain_Bypass: BOOL;
			Vacuum_Bypass: BOOL;
			Sealer_Bypass: BOOL;
			Stud_Bypass: BOOL;
			Turntable_Bypassed: BOOL;
			Door_Open: BOOL;

END_VAR

	(*data that needs to be retained in the event of a power cycle*)
	VAR PERSISTENT

		Load_Complete1: BOOL;
		Load_Complete2: BOOL;
		Load_Complete: BOOL;
		Stud_Complete: BOOL;
		Welding_Complete: BOOL;
		Sealing_Complete: BOOL;
		Unload_Complete: BOOL;
		TurnA_Complete: BOOL;
		TurnB_Complete: BOOL;
		Cycle_Complete: BOOL;
		Eject_Complete: BOOL;
		VacCheck_Complete: BOOL;
		Date_Stamp_Complete: BOOL;
		Load_Seq01: FB_GTAC_Load_Seq_20230302;
		Production_Count:INT;
		Repo_REQS: UINT;
		(*Allow_Load_PreCall: BOOL;
		Allow_Weld_PreCall: BOOL;
		Allow_Unload_PreCall: BOOL;*)
		(*All_SubPP_Off: BOOL;*)
		Production_Report: FB_Production_Report_20221007;

	END_VAR

	VAR_OUTPUT

		Prog_Ok: BOOL;
		Discrete_Image: udt_FixXX_Output_Image_20220715;
		In_Auto_Mode: BOOL;
		In_Manual_Mode: BOOL;
		Manual_Indicators1: DINT;
		Manual_Indicators2: DINT;
		Manual_Indicators3: DINT;
		At_Home: BOOL;
		Ready_To_Load: BOOL;
		Red_Lamp_Req: BOOL;
		Status: UINT;
		CLFaults1:UDINT;
		CLFaults2:UDINT;
		CLFaults3:UDINT;
		CLFaults4:UDINT;
		PPFaults: UDINT;
		PPFaults1: UDINT;
		PPFaults2: UDINT;
		Prod_Count_Out: INT;
		Cycle_Time_Out: TIME;
		PrevCycle_Time_Out: TIME;
		Load_Time_Out: TIME;
		Weld_Time_Out: TIME;
		Seal_Time_Out: TIME;
		Stud_Time_Out: TIME;
		Turn_Time_Out: TIME;
		Unload_Time_Out: TIME;
		Model_ID: UINT;
		TurntableA_At_Robot: BOOL;
		TurntableB_At_Robot: BOOL;
		Tool_Call_ForLoadRobots1: BOOL;
		Tool_Call_ForLoadRobots2: BOOL;
		Tool_Call_ForSealRobots: BOOL;
		Tool_Call_ForStudRobots: BOOL;
		Tool_Call_ForWeldRobots: BOOL;
		Tool_Call_ForSweepA: BOOL;
		Tool_Call_ForSweepB: BOOL;
		Tool_Call_ForUnloadRobots1: BOOL;
		Tool_Call_ForUnloadRobots2: BOOL;
		Robots_Clear_ToProceed: BOOL;
		Task_ID: UINT;
		Fix_ID: UINT;
		Load_Complete1_Ack: BOOL;
		Load_Complete2_Ack: BOOL;
		Seal_Complete_Ack: BOOL;
		Stud_Complete_Ack: BOOL;
		Weld_Complete_Ack: BOOL;
		TurnA_Complete_Ack: BOOL;
		TurnB_Complete_Ack: BOOL;
		Unload_Complete1_Ack: BOOL;
		Unload_Complete2_Ack: BOOL;
		Repo_Ack: UINT;
		Door_Close_Req: BOOL;
		Door_Open_Req: BOOL;
	END_VAR

	(*Set FB_OK to True*)
	Prog_OK:= TRUE;


	(*Set conditions to allow model change*)
	Fixture_Allow_Model_Change:= (In_Manual AND Tool_At_Home AND All_Sensors_Off AND All_Robots_Clear)
							OR (Model_ID=0);



(*$$$$$$$$$$$$$$$$$$$$$$$$$$$$$$$$$$$$$$$$$$$$ Fixture Bypasses $$$$$$$$$$$$$$$$$$$$$$$$$$$$$$$$$$$$$$$$$$$$$$$$$$$$*)
	Weld_Curtain_Bypass:= Discrete_In.Bypass_REQS.0;
	Vacuum_Bypass:= Discrete_In.Bypass_REQS.1;
	Stud_Bypass:= Discrete_In.Bypass_REQS.2;
	Turntable_Bypassed:= ((TurntableA_At_Robot AND Tool_At_Home AND All_Sensors_OFF)
					OR (Turntable_Bypassed AND NOT TurntableB_At_Robot))
					OR Discrete_In.Bypass_REQS.3;
	Sealer_Bypass:= MAIN.SL01.Disp1_Bypass;


(*$$$$$$$$$$$$$$$$$$$$$$$$$$$$$$$$$$$$$$$$$$$$ Gather Status Of Hardware $$$$$$$$$$$$$$$$$$$$$$$$$$$$$$$$$$$$$$$$$$$$$$$$$$$$*)
	(*Check on Status of Hardware*)
	Hardware();

(*$$$$$$$$$$$$$$$$$$$$$$$$$$$$$$$$$$$$$$$$$$$$$ Gather Standard Inputs $$$$$$$$$$$$$$$$$$$$$$$$$$$$$$$$$$$$$$$$$$$$$$$$$$$$$$$$$*)

(*Clamp/Cylinder Inputs*)
	Cylinders();

(*Part Present Inputs*)
	Proxies();

(*$$$$$$$$$$$$$$$$$$$$$$$$$$$$$$$$$$$$$$$$$$$ Qaulity Checking Routines $$$$$$$$$$$$$$$$$$$$$$$$$$$$$$$$$$$$$$$$$$$$$$$$$$$$$$$$$*)

	(*QA Checks*)
		CheckQA1FB(
			Start_QAcheck:= Auto_Run AND Enable_Motion AND Tool_At_Load.3,
			QAcheck_Reset:= Cycle_Complete OR (In_Manual AND Discrete_In.Go_Home AND All_Sensors_Off),
			QAcheck_Retry:= In_From_ICxx.QA_Reset.0,
			QAcheck_Release:= In_From_ICxx.QA_Reset.1,
			QAcheck_Adv_In:= QACheck1ADVD AND QACheck2ADVD,
			QAcheck_Ret_In:= QACheck1RETD AND QACheck2RETD,
			User_Dry_Cycle:= Dry_Cycle,
			QAcheck_OK_Delay:= T#0.75s,
			QAcheck_Fault_Delay:= T#3.0s,
			QAcheck_OK=> All_QAChecks_OK,
			QAcheck_Failed=> QAChecks_Failed);



(*$$$$$$$$$$$$$$$$$$$$$$$$$$$$$$$$$$$$$$$$$$$$$$$$ Internal Code $$$$$$$$$$$$$$$$$$$$$$$$$$$$$$$$$$$$$$$$$$$$$$$$$$$$$$$$$$$$$$$$$$$$*)
(*Auto / Manual Mode Code*)
	IF Discrete_In.Mode_Select.0 AND NOT Discrete_In.Mode_Select.1
		THEN
			In_Auto:= TRUE;
			In_Auto_Mode:= TRUE;
	END_IF;
	IF NOT Discrete_In.Mode_Select.0 AND Discrete_In.Mode_Select.1
		THEN
			In_Auto:= FALSE;
			In_Auto_Mode:= FALSE;
	END_IF;
	In_Manual:= NOT In_Auto;
	In_Manual_Mode:= In_Manual;

(*--------------------------------------------------------------------------------Tool Positions---------------------------------------------------------------*)
	Tool_States();

(*----------------------------------------------------Part Present Sensor Input Patterns----------------------------------------------------------------*)
	All_Sensors();


(*>>>>>>>>>>>>>>>>>>>>>>>>>>>>>>>>>>>>>>>>>> Auto Run Cycle >>>>>>>>>>>>>>>>>>>>>>>>>>>>>>>>>>>>>>>*)
(*+++++++++++THIS AREA IS CUSTOM PER INSTALLATION AND WILL HAVE TO BE MODIFIED PER +++++++++++++*)
(*+++++++++++THIS AREA IS CUSTOM PER INSTALLATION AND WILL HAVE TO BE MODIFIED PER +++++++++++++*)
	(*Control of Auto_Run*)
	Auto_Run:= Enable_Motion AND In_Auto AND Model_ID<>0 AND NOT Cycle_Complete;

	(*Auto Run Enables All Other Auto Cycle Code*)
	IF Auto_Run
		THEN

			IF (NOT Load_Complete1 OR (Load_Robots_UnclampEarly1 AND All_Sensors_On.1))
				AND Load_Robots_Clear2 AND Stud_Robots_Clear AND Seal_Robots_Clear
				AND Weld_Robots_Clear AND TurnTable_Clear AND Unload_Robots_Clear
				AND TurnTableA_At_Robot
				THEN
					(*Start 1st Load Robots*)
					Start_Load_Robots1:= ((Tool_At_Load.0 AND All_Sensors_Off AND NOT Repo_Reqs.0 AND Load_Robots_PartInEOAT1)
									OR (Tool_At_Load.1 AND All_Sensors_On.4 AND Repo_Reqs.0))
									OR Load_Robots_WorkingOK1;
					(*Allow 1st Load Robots To Proceed*)
					Load_Robots_Proceed1:= Tool_At_Load.0 AND All_Sensors_Off AND Load_Robots_PartInEOAT1;
			ELSE
					Start_Load_Robots1:= FALSE;
					Load_Robots_Proceed1:= FALSE;
			END_IF;


			IF (NOT Load_Complete2 OR (Load_Robots_UnclampEarly2 AND All_Sensors_On.2))
				AND Load_Robots_Clear1 AND Stud_Robots_Clear AND Seal_Robots_Clear
				AND Weld_Robots_Clear AND TurnTable_Clear AND Unload_Robots_Clear
				AND TurnTableA_At_Robot
				THEN
					(*Start 2nd Load Robots*)
					Start_Load_Robots2:= ((Tool_At_Load.1 AND All_Sensors_Off AND NOT Repo_Reqs.0 AND Load_Robots_PartInEOAT2)
									OR (Tool_At_Load.1 AND All_Sensors_On.4 AND Repo_Reqs.0))
									OR Load_Robots_WorkingOK2;
					(*Allow 2nd Load Robots To Proceed*)
					Load_Robots_Proceed2:= Tool_At_Load.1 AND All_Sensors_Off AND Load_Robots_PartInEOAT2;
			ELSE
					Start_Load_Robots2:= FALSE;
					Load_Robots_Proceed2:= FALSE;
			END_IF;


			IF NOT Sealer_Bypass AND Load_Complete AND NOT Sealing_Complete
				AND Load_Robots_Clear AND Stud_Robots_Clear AND  Weld_Robots_Clear AND TurnTable_Clear AND Unload_Robots_Clear
				AND TurnTableA_At_Robot
				THEN
					(*Start Seal Robots*)
					Start_Seal_Robots:= ((Tool_At_Seal.0 AND All_Sensors_On.3 AND NOT Repo_Reqs.1 AND NOT MAIN.SL01.Disp1_Faulted AND MAIN.SL01.Disp1_Ready)
									OR (Tool_At_Seal.1 AND All_Sensors_On.4 AND Repo_Reqs.1))
									OR Seal_Robots_WorkingOK;
					(*Allow Seal Robots To Proceed*)
					Seal_Robots_Proceed:= Tool_At_Seal.0 AND All_Sensors_On.3;
			ELSE
					Start_Seal_Robots:= FALSE;
					Seal_Robots_Proceed:= FALSE;
			END_IF;


			IF NOT Stud_Bypass AND Load_Complete AND NOT Stud_Complete AND NOT Welding_Complete
				AND Load_Robots_Clear AND Seal_Robots_Clear AND  Weld_Robots_Clear AND TurnTable_Clear AND Unload_Robots_Clear
				AND TurnTableA_At_Robot
				THEN
					(*Start Stud Robots*)
					Start_Stud_Robots:= ((Tool_At_Stud.0 AND All_Sensors_On.3 AND NOT Repo_Reqs.2)
									OR (Tool_At_Stud.1 AND All_Sensors_On.4 AND Repo_Reqs.2))
									OR Stud_Robots_WorkingOK;
					(*Allow Stud Robots To Proceed*)
					Stud_Robots_Proceed:= Tool_At_Stud.0 AND All_Sensors_On.3;
			ELSE
					Start_Stud_Robots:= FALSE;
					Stud_Robots_Proceed:= FALSE;
			END_IF;


                             IF  NOT TurnA_Complete AND Load_Complete AND NOT Welding_Complete AND NOT Unload_Complete
				 AND Load_Robots_Clear AND Seal_Robots_Clear AND Stud_Robots_Clear AND  Weld_Robots_Clear AND Unload_Robots_Clear
				AND (NOT TurntableA_At_Robot OR TurnTable_WorkingOK)
				THEN
					(*Start Turntable SweepA (Fix01 to the Robot)*)
					Start_TurntableA:= ((Tool_At_Rotate.0 AND All_Sensors_On.3)
									OR (All_Sensors_Off AND Tool_At_Home))
									OR TurnTable_WorkingOK;
			ELSE
					Start_TurntableA:= FALSE;
			END_IF;


			IF NOT TurnB_Complete AND Welding_Complete AND NOT Unload_Complete AND (Sealing_Complete OR Sealer_Bypass) AND (Stud_Complete OR Stud_Bypass)
				AND Load_Robots_Clear AND Seal_Robots_Clear AND Stud_Robots_Clear AND Weld_Robots_Clear  AND Unload_Robots_Clear
				AND (NOT TurntableB_At_Robot OR TurnTable_WorkingOK)
				THEN
					(*Start Turntable SweepB (Fix01 to the Operator)*)
					Start_TurntableB:= TRUE;
                             ELSIF All_Sensors_Off AND NOT TurnB_Complete AND Weld_Robots_Clear AND Load_Robots_Clear AND Unload_Robots_Clear
				AND (NOT TurntableB_At_Robot OR TurnTable_WorkingOK)
			THEN
					Start_TurntableB:= All_Sensors_Off;
                             ELSE
					Start_TurntableB:= FALSE;
                             END_IF;


			IF Load_Complete AND NOT Welding_Complete AND (Sealing_Complete OR Sealer_Bypass) AND (Stud_Complete OR Stud_Bypass) AND NOT Unload_Complete
				AND Load_Robots_Clear AND Seal_Robots_Clear AND Stud_Robots_Clear AND TurnTable_Clear AND Unload_Robots_Clear
				AND TurnTableA_At_Robot AND Mig_Robots_Ready 
				THEN
					(*Start Weld Robots*)
					Start_Weld_Robots:=((Tool_At_Weld.0 AND NOT Repo_Reqs.3 AND NOT Repo_Reqs.4 AND NOT Repo_Reqs.5 AND All_Sensors_On.3)
										OR (Tool_At_Weld.1 AND Repo_Reqs.3 AND All_Sensors_On.3)
										OR (Tool_At_Weld.2 AND Repo_Reqs.4 AND All_Sensors_On.4)
										OR (Tool_At_Weld.3 AND Repo_Reqs.5 AND All_Sensors_On.5)
										OR (Tool_At_Unload.0 AND Weld_Robots_UnclampEarly))
										OR Weld_Robots_WorkingOK;
					(*Allow Weld Robots To Proceed*)
					Weld_Robots_Proceed:= Load_Complete AND Tool_At_Weld.0 AND All_Sensors_On.3;
			ELSE
					Start_Weld_Robots:= FALSE;
					Weld_Robots_Proceed:= FALSE;
			END_IF;


			IF Welding_Complete  AND (Sealing_Complete OR Sealer_Bypass) AND (Stud_Complete OR Stud_Bypass) AND NOT Unload_Complete
				AND Load_Robots_Clear AND Seal_Robots_Clear AND Stud_Robots_Clear AND TurnTable_Clear AND Unload_Robots_Clear2
				AND TurnTableA_At_Robot
				THEN
					(*Start Unload Robots*)
					Start_Unload_Robots1:=((((Tool_At_Unload.0 AND NOT Repo_Reqs.6 AND NOT Repo_Reqs.7 AND All_Sensors_On.8)
										OR (Tool_At_Unload.1 AND Repo_Reqs.6)
										OR (Tool_At_Unload.2 AND Repo_Reqs.7))
										AND (All_Sensors_On.8 AND Unload_Robots_EOATEmpty1))
										OR (NOT Unload_Robots_Clear1 AND NOT Unload_Robots_EOATEmpty1))
										OR Unload_Robots_WorkingOK1;
					(*Allow Unload Robots To Proceed*)
					Unload_Robots_Proceed1:= Welding_Complete AND Tool_At_Unload.0 AND All_Sensors_On.8 AND Unload_Robots_EOATEmpty1;
			ELSE
					Start_Unload_Robots1:= FALSE;
					Unload_Robots_Proceed1:= FALSE;
			END_IF;


			IF Welding_Complete  AND (Sealing_Complete OR Sealer_Bypass) AND (Stud_Complete OR Stud_Bypass) AND NOT Unload_Complete
				AND Load_Robots_Clear AND Seal_Robots_Clear AND Stud_Robots_Clear AND TurnTable_Clear AND Unload_Robots_Clear1
				AND TurnTableA_At_Robot
				THEN
					(*Start Unload Robots*)
					Start_Unload_Robots2:=((((Tool_At_Unload.0 AND NOT Repo_Reqs.6 AND NOT Repo_Reqs.7 AND All_Sensors_On.8)
										OR (Tool_At_Unload.1 AND Repo_Reqs.6)
										OR (Tool_At_Unload.2 AND Repo_Reqs.7))
										AND (All_Sensors_On.8 AND Unload_Robots_EOATEmpty2))
										OR (NOT Unload_Robots_Clear2 AND NOT Unload_Robots_EOATEmpty2))
										OR Unload_Robots_WorkingOK2;
					(*Allow Unload Robots To Proceed*)
					Unload_Robots_Proceed2:= Welding_Complete AND Tool_At_Unload.0 AND All_Sensors_On.8 AND Unload_Robots_EOATEmpty2;
			ELSE
					Start_Unload_Robots2:= FALSE;
					Unload_Robots_Proceed2:= FALSE;
			END_IF;


	ELSE
		Start_Load_Robots1:= FALSE;
		Start_Load_Robots2:= FALSE;
		Start_Seal_Robots:= FALSE;
		Start_Stud_Robots:= FALSE;
		Start_TurntableA:= FALSE;
		Start_TurntableB:= FALSE;
		Start_Weld_Robots:= FALSE;
		Start_Unload_Robots1:= FALSE;
		Start_Unload_Robots2:= FALSE;
		Load_Robots_Proceed1:=FALSE;
		Load_Robots_Proceed2:=FALSE;
		Seal_Robots_Proceed:=FALSE;
		Weld_Robots_Proceed:=FALSE;
		Unload_Robots_Proceed1:=FALSE;
		Unload_Robots_Proceed2:=FALSE;
	END_IF;




(*---------------------------------------------------------------Completes----------------------------------------------------*)
	(*1st Load Complete*)
	IF NOT Dry_Cycle
		THEN
		Load_Complete1:=  All_Sensors_On.1;
	ELSIF Dry_Cycle
		THEN
		IF Tool_At_Home AND Enable_Motion AND All_Sensors_Off
			THEN
			Load_Complete1:= TRUE;
		END_IF;
	END_IF;
	(*2nd Load Complete*)
	IF NOT Dry_Cycle
		THEN
		Load_Complete2:=  All_Sensors_On.2;
	ELSIF Dry_Cycle
		THEN
		IF Tool_At_Home AND Enable_Motion AND All_Sensors_Off
			THEN
			Load_Complete2:= TRUE;
		END_IF;
	END_IF;
	(*All Load Complete*)
	IF NOT Dry_Cycle
		THEN
		Load_Complete:= (All_Sensors_On.2
					OR (All_Sensors_On.3 AND Tool_At_Weld.0)
					OR (Repo_Reqs.0 AND All_Sensors_On.4)
					OR (Repo_Reqs.1 AND All_Sensors_On.5)
					OR (Repo_Reqs.2 AND All_Sensors_On.6))
					OR Weld_Robots_WorkingOK OR Welding_Complete;
	ELSIF Dry_Cycle
		THEN
		IF Load_Complete1 AND Load_Complete2 AND All_Sensors_Off
			THEN
			Load_Complete:= TRUE;
		END_IF;
	END_IF;

	(*Welding Complete*)
	IF Weld_Robots_Complete
		THEN
		Welding_Complete:= TRUE;
	END_IF;

	(*Unload Complete*)
	IF NOT Dry_Cycle
		THEN
			IF (Unload_Robots_Complete1 OR Unload_Robots_Complete2 OR (All_Sensors_Off AND Unload_Robots_Clear)) AND Welding_Complete
				THEN
				Unload_Complete:= TRUE;
			END_IF;
	ELSIF Dry_Cycle
		THEN
			IF (Unload_Robots_Complete1 OR Unload_Robots_Complete2 OR (All_Sensors_Off AND Unload_Robots_Clear)) AND Welding_Complete
				THEN
				Unload_Complete:= TRUE;
			END_IF;
	END_IF;
(*!!!!!!!!!!!!!!!!!!!!!!!!!!!!!!!!!!!!!!!!!!!!!!!!!!!!!!!!!!!!!!!!!!!!!!!!!!!!!!!!!!!!!!!!!!!!!!!!! Cycle Complete !!!!!!!!!!!!!!!!!!!!!!!!!!!!!!!!!!!!!!!!!!!!!!!!!!!!!!!!!!!!!!!!!!!!!!!!!!!!!!!!!!!!!!!!!!*)
	(*Set Cycle Complete*)
	IF Auto_Run AND Load_Complete AND Welding_Complete AND Unload_Complete AND All_Robots_Clear
		THEN Cycle_Complete:= TRUE;
	END_IF;
	(*Reset All Completes*)
	IF Load_Robots_Clear AND Weld_Robots_Clear AND Unload_Robots_Clear AND NOT Unload_Robots_Complete1 AND NOT Unload_Robots_Complete2
		THEN
			IF In_Manual AND Discrete_In.Go_Home AND All_Sensors_Off
				THEN
					Reset_All_Completes:= TRUE;
			ELSIF NOT Dry_Cycle AND Cycle_Complete AND NOT Enable_Motion AND Tool_At_Home AND All_Sensors_Off
				THEN
					Reset_All_Completes:= TRUE;
			ELSIF Dry_Cycle AND Cycle_Complete AND Tool_At_Home AND All_Sensors_Off
				THEN
					Reset_All_Completes:=TRUE;
			ELSE
					Reset_All_Completes:= FALSE;
			END_IF;
	END_IF;
	(*Perform Actual Reset*)
		IF Reset_All_Completes
			THEN
				Cycle_Complete:= FALSE;
				Load_Complete1:= FALSE;
				Load_Complete2:= FALSE;
				Load_Complete:= FALSE;
				Sealing_Complete:= FALSE;
				Stud_Complete:= FALSE;
				Welding_Complete:= FALSE;
				Date_Stamp_Complete:= FALSE;
				VacCheck_Complete:= FALSE;
				Unload_Complete:=FALSE;
				Eject_Complete:= FALSE;
				Load_Robots_UnclampEarly1:= FALSE;
				Load_Robots_UnclampEarly2:= FALSE;
				Seal_Robots_UnclampEarly:= FALSE;
				Stud_Robots_UnclampEarly:= FALSE;
				Weld_Robots_UnclampEarly:= FALSE;
				Repo_Reqs:= 0;
				Reset_All_Completes:= FALSE;

		END_IF;

(*---------------------------------------------------------------------------- Call Various Actions ----------------------------------------------------------------------------------------------------*)
	(*Poduction Counters and Report*)
	Production();

	(*Register Robot(s) to Fixture*)
	Robot_Registration();

	(*Setup Fix ID and Model Data*)
	Task_Fix_Model_IDs();

	(*Generate Status Banner and Fault Flags*)
	Status_and_Faults();

	(*Tool Clamp / Unclamp Sequencing and Reposition Handling*)
	Tool_VBSeq_Repos();

	(*Transfer Object Image Data to UI Section*)
	Xfer_To_UI();


(*-----------------------------------------------------------------------------------------Transfer Valve Outputs --------------------------------------------------------------------------------*)
	(*Move "Manual_Home_Prompt" as required for home prompting*)
		Manual_Ind_HomePrompt:= Flash_Rate AND In_Manual AND Discrete_In.Go_Home AND NOT Tool_At_Home;

	(*Call each valve bank*)
	ValveBank1();
	(*ValveBank2();
	ValveBank3(); *)

	(*Door Close Request*)
		Door_Close_Req:= NOT Weld_Curtain_Bypass AND (In_Auto AND TurntableB_At_Robot AND Enable_Motion
					AND NOT CLFaulted.0 AND NOT PPFaulted.0 AND NOT QAChecks_Failed
					AND ((Load_Complete AND NOT Welding_Complete) OR (Enable_Motion AND TurnTable_Bypassed) OR Dry_Cycle))
					OR (In_Manual AND MAIN.IC01.OP1_LC_Clear AND Discrete_In.CustomApplication_REQS.7);

	(*Door Open Request*)
		Door_Open_Req:= Weld_Curtain_Bypass OR (NOT Dry_Cycle AND TurntableB_At_Robot AND In_Auto AND All_Robots_Clear
					AND ((Welding_Complete AND NOT Dry_Cycle)
					OR (NOT Welding_Complete AND (CLFaulted.0 OR PPFaulted.0 OR QAChecks_Failed))
					OR (Tool_At_Home AND All_Sensors_Off AND NOT Turntable_Bypassed)))
					OR (In_Manual AND  (Discrete_In.CustomApplication_REQS.6 OR (TurntableB_At_Robot AND Discrete_In.Go_Home)));

ACTION All_Sensors:


(*+++++++++++THIS AREA IS CUSTOM PER INSTALLATION AND WILL HAVE TO BE MODIFIED PER +++++++++++++*)
(*+++++++++++THIS AREA IS CUSTOM PER INSTALLATION AND WILL HAVE TO BE MODIFIED PER +++++++++++++*)
(*+++++++++++THIS AREA IS CUSTOM PER INSTALLATION AND WILL HAVE TO BE MODIFIED PER +++++++++++++*)



(**************************************************************************All Sensors Off******************************************************************************)
(**************************************************************************All Sensors Off******************************************************************************)
(**************************************************************************All Sensors Off******************************************************************************)

	(*All Sensors Required Off*)
	All_Sensors_Off:= NOT Part_Present1 AND NOT Part_Present2 AND NOT  Part_Present3
			AND NOT Part_Present4 AND NOT Part_Present5 AND NOT Part_Present6
			AND NOT Part_Present7 AND NOT Part_Present8 AND NOT Part_Present9
			AND NOT Part_Present10 AND NOT Part_Present11 AND NOT Part_Present12
			AND NOT Part_Present13 AND NOT Part_Present14 AND NOT Part_Present15
			AND NOT Part_Present16 AND NOT Part_Present17 AND NOT Part_Present18
			AND NOT Part_Present19 AND NOT Part_Present20 AND NOT Part_Present21
			AND NOT Part_Present22 AND NOT Part_Present23 AND NOT Part_Present24
			AND NOT Part_Present25 AND NOT Part_Present26 AND NOT Part_Present27
			AND NOT Part_Present28 AND NOT Part_Present29 AND NOT Part_Present30
			AND NOT Part_Present31 AND NOT Part_Present32 AND NOT Part_Present33
			AND NOT Part_Present34 AND NOT Part_Present35 AND NOT Part_Present36
			AND NOT Part_Present37 AND NOT Part_Present38 AND NOT Part_Present39
			AND NOT Part_Present40;

	(*All Sensors Required Off - Used for sub fixtures where the part has to move from one stage to the next*)
	All_Sensors_Off1:= NOT Part_Present1 AND NOT Part_Present2 AND NOT  Part_Present3
			AND NOT Part_Present4 AND NOT Part_Present5 AND NOT Part_Present6
			AND NOT Part_Present7 AND NOT Part_Present8 AND NOT Part_Present9
			AND NOT Part_Present10 AND NOT Part_Present11 AND NOT Part_Present12
			AND NOT Part_Present13 AND NOT Part_Present14 AND NOT Part_Present15
			AND NOT Part_Present16 AND NOT Part_Present17 AND NOT Part_Present18
			AND NOT Part_Present19 AND NOT Part_Present20 AND NOT Part_Present21
			AND NOT Part_Present22 AND NOT Part_Present23 AND NOT Part_Present24
			AND NOT Part_Present25 AND NOT Part_Present26 AND NOT Part_Present27
			AND NOT Part_Present28 AND NOT Part_Present29 AND NOT Part_Present30
			AND NOT Part_Present31 AND NOT Part_Present32 AND NOT Part_Present33
			AND NOT Part_Present34 AND NOT Part_Present35 AND NOT Part_Present36
			AND NOT Part_Present37 AND NOT Part_Present38 AND NOT Part_Present39
			AND NOT Part_Present40;

	(*All Sensors Required Off - Used for sub fixtures where the part has to move from one stage to the next*)
	All_Sensors_Off2:= NOT Part_Present1 AND NOT Part_Present2 AND NOT  Part_Present3
			AND NOT Part_Present4 AND NOT Part_Present5 AND NOT Part_Present6
			AND NOT Part_Present7 AND NOT Part_Present8 AND NOT Part_Present9
			AND NOT Part_Present10 AND NOT Part_Present11 AND NOT Part_Present12
			AND NOT Part_Present13 AND NOT Part_Present14 AND NOT Part_Present15
			AND NOT Part_Present16 AND NOT Part_Present17 AND NOT Part_Present18
			AND NOT Part_Present19 AND NOT Part_Present20 AND NOT Part_Present21
			AND NOT Part_Present22 AND NOT Part_Present23 AND NOT Part_Present24
			AND NOT Part_Present25 AND NOT Part_Present26 AND NOT Part_Present27
			AND NOT Part_Present28 AND NOT Part_Present29 AND NOT Part_Present30
			AND NOT Part_Present31 AND NOT Part_Present32 AND NOT Part_Present33
			AND NOT Part_Present34 AND NOT Part_Present35 AND NOT Part_Present36
			AND NOT Part_Present37 AND NOT Part_Present38 AND NOT Part_Present39
			AND NOT Part_Present40;



(**************************************************************************All Sensors On******************************************************************************)
(**************************************************************************All Sensors On******************************************************************************)
(**************************************************************************All Sensors On******************************************************************************)


	(*Sensors Required for Start Of 1st Robot Load*)
	All_Sensors_On.0:= FALSE OR (Dry_Cycle AND All_Sensors_Off);
	(*Sensors Required for Start of 2nd Robot Load*)
	All_Sensors_On.1:= FALSE OR  (Dry_Cycle AND All_Sensors_Off);

	(*Sensors After Load Complete*)
	All_Sensors_On.2:=(
					((Model_ID=1)
						AND Part_Present1 AND Part_Present2 AND Part_Present3
						AND Part_Present4 AND Part_Present5 AND Part_Present6
						AND Part_Present7 AND Part_Present8 AND Part_Present9
						AND Part_Present10 AND Part_Present11 AND Part_Present12
						AND Part_Present13 AND Part_Present14 AND Part_Present15
						AND Part_Present16 AND Part_Present17 AND Part_Present18
						AND Part_Present19 AND Part_Present20 AND Part_Present21
						AND Part_Present22 AND Part_Present23 AND Part_Present24
						AND Part_Present25 AND Part_Present26 AND Part_Present27
						AND Part_Present28 AND Part_Present29 AND Part_Present30
						AND Part_Present31 AND Part_Present32 AND Part_Present33
						AND Part_Present34 AND Part_Present35 AND Part_Present36
						AND Part_Present37 AND Part_Present38 AND Part_Present39
						AND Part_Present40)

					OR ((Model_ID=2)
						AND Part_Present1 AND Part_Present2 AND Part_Present3
						AND Part_Present4 AND Part_Present5 AND Part_Present6
						AND Part_Present7 AND Part_Present8 AND Part_Present9
						AND Part_Present10 AND Part_Present11 AND Part_Present12
						AND Part_Present13 AND Part_Present14 AND Part_Present15
						AND Part_Present16 AND Part_Present17 AND Part_Present18
						AND Part_Present19 AND Part_Present20 AND Part_Present21
						AND Part_Present22 AND Part_Present23 AND Part_Present24
						AND Part_Present25 AND Part_Present26 AND Part_Present27
						AND Part_Present28 AND Part_Present29 AND Part_Present30
						AND Part_Present31 AND Part_Present32 AND Part_Present33
						AND Part_Present34 AND Part_Present35 AND Part_Present36
						AND Part_Present37 AND Part_Present38 AND Part_Present39
						AND Part_Present40)

					OR ((Model_ID=3)
						AND Part_Present1 AND Part_Present2 AND Part_Present3
						AND Part_Present4 AND Part_Present5 AND Part_Present6
						AND Part_Present7 AND Part_Present8 AND Part_Present9
						AND Part_Present10 AND Part_Present11 AND Part_Present12
						AND Part_Present13 AND Part_Present14 AND Part_Present15
						AND Part_Present16 AND Part_Present17 AND Part_Present18
						AND Part_Present19 AND Part_Present20 AND Part_Present21
						AND Part_Present22 AND Part_Present23 AND Part_Present24
						AND Part_Present25 AND Part_Present26 AND Part_Present27
						AND Part_Present28 AND Part_Present29 AND Part_Present30
						AND Part_Present31 AND Part_Present32 AND Part_Present33
						AND Part_Present34 AND Part_Present35 AND Part_Present36
						AND Part_Present37 AND Part_Present38 AND Part_Present39
						AND Part_Present40)

					OR ((Model_ID=4)
						AND Part_Present1 AND Part_Present2 AND Part_Present3
						AND Part_Present4 AND Part_Present5 AND Part_Present6
						AND Part_Present7 AND Part_Present8 AND Part_Present9
						AND Part_Present10 AND Part_Present11 AND Part_Present12
						AND Part_Present13 AND Part_Present14 AND Part_Present15
						AND Part_Present16 AND Part_Present17 AND Part_Present18
						AND Part_Present19 AND Part_Present20 AND Part_Present21
						AND Part_Present22 AND Part_Present23 AND Part_Present24
						AND Part_Present25 AND Part_Present26 AND Part_Present27
						AND Part_Present28 AND Part_Present29 AND Part_Present30
						AND Part_Present31 AND Part_Present32 AND Part_Present33
						AND Part_Present34 AND Part_Present35 AND Part_Present36
						AND Part_Present37 AND Part_Present38 AND Part_Present39
						AND Part_Present40)
					) OR (All_Sensors_Off AND Dry_Cycle);


	(*Sensors Require for Start Of Welding*)
	All_Sensors_On.3:=(
					((Model_ID=1)
						AND Part_Present1 AND Part_Present2 AND Part_Present3
						AND Part_Present4 AND Part_Present5 AND Part_Present6
						AND Part_Present7 AND Part_Present8 AND Part_Present9
						AND Part_Present10 AND Part_Present11 AND Part_Present12
						AND Part_Present13 AND Part_Present14 AND Part_Present15
						AND Part_Present16 AND Part_Present17 AND Part_Present18
						AND Part_Present19 AND Part_Present20 AND Part_Present21
						AND Part_Present22 AND Part_Present23 AND Part_Present24
						AND Part_Present25 AND Part_Present26 AND Part_Present27
						AND Part_Present28 AND Part_Present29 AND Part_Present30
						AND Part_Present31 AND Part_Present32 AND Part_Present33
						AND Part_Present34 AND Part_Present35 AND Part_Present36
						AND Part_Present37 AND Part_Present38 AND Part_Present39
						AND Part_Present40)

					OR ((Model_ID=2)
						AND Part_Present1 AND Part_Present2 AND Part_Present3
						AND Part_Present4 AND Part_Present5 AND Part_Present6
						AND Part_Present7 AND Part_Present8 AND Part_Present9
						AND Part_Present10 AND Part_Present11 AND Part_Present12
						AND Part_Present13 AND Part_Present14 AND Part_Present15
						AND Part_Present16 AND Part_Present17 AND Part_Present18
						AND Part_Present19 AND Part_Present20 AND Part_Present21
						AND Part_Present22 AND Part_Present23 AND Part_Present24
						AND Part_Present25 AND Part_Present26 AND Part_Present27
						AND Part_Present28 AND Part_Present29 AND Part_Present30
						AND Part_Present31 AND Part_Present32 AND Part_Present33
						AND Part_Present34 AND Part_Present35 AND Part_Present36
						AND Part_Present37 AND Part_Present38 AND Part_Present39
						AND Part_Present40)

					OR ((Model_ID=3)
						AND Part_Present1 AND Part_Present2 AND Part_Present3
						AND Part_Present4 AND Part_Present5 AND Part_Present6
						AND Part_Present7 AND Part_Present8 AND Part_Present9
						AND Part_Present10 AND Part_Present11 AND Part_Present12
						AND Part_Present13 AND Part_Present14 AND Part_Present15
						AND Part_Present16 AND Part_Present17 AND Part_Present18
						AND Part_Present19 AND Part_Present20 AND Part_Present21
						AND Part_Present22 AND Part_Present23 AND Part_Present24
						AND Part_Present25 AND Part_Present26 AND Part_Present27
						AND Part_Present28 AND Part_Present29 AND Part_Present30
						AND Part_Present31 AND Part_Present32 AND Part_Present33
						AND Part_Present34 AND Part_Present35 AND Part_Present36
						AND Part_Present37 AND Part_Present38 AND Part_Present39
						AND Part_Present40)

					OR ((Model_ID=4)
						AND Part_Present1 AND Part_Present2 AND Part_Present3
						AND Part_Present4 AND Part_Present5 AND Part_Present6
						AND Part_Present7 AND Part_Present8 AND Part_Present9
						AND Part_Present10 AND Part_Present11 AND Part_Present12
						AND Part_Present13 AND Part_Present14 AND Part_Present15
						AND Part_Present16 AND Part_Present17 AND Part_Present18
						AND Part_Present19 AND Part_Present20 AND Part_Present21
						AND Part_Present22 AND Part_Present23 AND Part_Present24
						AND Part_Present25 AND Part_Present26 AND Part_Present27
						AND Part_Present28 AND Part_Present29 AND Part_Present30
						AND Part_Present31 AND Part_Present32 AND Part_Present33
						AND Part_Present34 AND Part_Present35 AND Part_Present36
						AND Part_Present37 AND Part_Present38 AND Part_Present39
						AND Part_Present40)
					) OR (All_Sensors_Off AND Dry_Cycle);


	(*Sensors Required After Repo_Reqs.0*)
	All_Sensors_On.4:= (FALSE) OR (Dry_Cycle AND All_Sensors_Off);
	(*Sensors Required After Repo_Reqs.1*)
	All_Sensors_On.5:= (FALSE) OR (Dry_Cycle AND All_Sensors_Off);
	(*Sensors Required After Repo_Reqs.2*)
	All_Sensors_On.6:= (FALSE) OR (Dry_Cycle AND All_Sensors_Off);
	(*Sensors Required After Repo_Reqs.3*)
	All_Sensors_On.7:= (FALSE) OR (Dry_Cycle AND All_Sensors_Off);


	(*Sensors Required for Start Of Unload1*)
	All_Sensors_On.8:=(
					((Model_ID=1)
						AND Part_Present1 AND Part_Present2 AND Part_Present3
						AND Part_Present4 AND Part_Present5 AND Part_Present6
						AND Part_Present7 AND Part_Present8 AND Part_Present9
						AND Part_Present10 AND Part_Present11 AND Part_Present12
						AND Part_Present13 AND Part_Present14 AND Part_Present15
						AND Part_Present16 AND Part_Present17 AND Part_Present18
						AND Part_Present19 AND Part_Present20 AND Part_Present21
						AND Part_Present22 AND Part_Present23 AND Part_Present24
						AND Part_Present25 AND Part_Present26 AND Part_Present27
						AND Part_Present28 AND Part_Present29 AND Part_Present30
						AND Part_Present31 AND Part_Present32 AND Part_Present33
						AND Part_Present34 AND Part_Present35 AND Part_Present36
						AND Part_Present37 AND Part_Present38 AND Part_Present39
						AND Part_Present40)

					OR ((Model_ID=2)
						AND Part_Present1 AND Part_Present2 AND Part_Present3
						AND Part_Present4 AND Part_Present5 AND Part_Present6
						AND Part_Present7 AND Part_Present8 AND Part_Present9
						AND Part_Present10 AND Part_Present11 AND Part_Present12
						AND Part_Present13 AND Part_Present14 AND Part_Present15
						AND Part_Present16 AND Part_Present17 AND Part_Present18
						AND Part_Present19 AND Part_Present20 AND Part_Present21
						AND Part_Present22 AND Part_Present23 AND Part_Present24
						AND Part_Present25 AND Part_Present26 AND Part_Present27
						AND Part_Present28 AND Part_Present29 AND Part_Present30
						AND Part_Present31 AND Part_Present32 AND Part_Present33
						AND Part_Present34 AND Part_Present35 AND Part_Present36
						AND Part_Present37 AND Part_Present38 AND Part_Present39
						AND Part_Present40)

					OR ((Model_ID=3)
						AND Part_Present1 AND Part_Present2 AND Part_Present3
						AND Part_Present4 AND Part_Present5 AND Part_Present6
						AND Part_Present7 AND Part_Present8 AND Part_Present9
						AND Part_Present10 AND Part_Present11 AND Part_Present12
						AND Part_Present13 AND Part_Present14 AND Part_Present15
						AND Part_Present16 AND Part_Present17 AND Part_Present18
						AND Part_Present19 AND Part_Present20 AND Part_Present21
						AND Part_Present22 AND Part_Present23 AND Part_Present24
						AND Part_Present25 AND Part_Present26 AND Part_Present27
						AND Part_Present28 AND Part_Present29 AND Part_Present30
						AND Part_Present31 AND Part_Present32 AND Part_Present33
						AND Part_Present34 AND Part_Present35 AND Part_Present36
						AND Part_Present37 AND Part_Present38 AND Part_Present39
						AND Part_Present40)

					OR ((Model_ID=4)
						AND Part_Present1 AND Part_Present2 AND Part_Present3
						AND Part_Present4 AND Part_Present5 AND Part_Present6
						AND Part_Present7 AND Part_Present8 AND Part_Present9
						AND Part_Present10 AND Part_Present11 AND Part_Present12
						AND Part_Present13 AND Part_Present14 AND Part_Present15
						AND Part_Present16 AND Part_Present17 AND Part_Present18
						AND Part_Present19 AND Part_Present20 AND Part_Present21
						AND Part_Present22 AND Part_Present23 AND Part_Present24
						AND Part_Present25 AND Part_Present26 AND Part_Present27
						AND Part_Present28 AND Part_Present29 AND Part_Present30
						AND Part_Present31 AND Part_Present32 AND Part_Present33
						AND Part_Present34 AND Part_Present35 AND Part_Present36
						AND Part_Present37 AND Part_Present38 AND Part_Present39
						AND Part_Present40)
					) OR (All_Sensors_Off AND Dry_Cycle);

	(*Sensors Required for Start Of Unload2*)
	All_Sensors_On.9:=(
					((Model_ID=1)
						AND Part_Present1 AND Part_Present2 AND Part_Present3
						AND Part_Present4 AND Part_Present5 AND Part_Present6
						AND Part_Present7 AND Part_Present8 AND Part_Present9
						AND Part_Present10 AND Part_Present11 AND Part_Present12
						AND Part_Present13 AND Part_Present14 AND Part_Present15
						AND Part_Present16 AND Part_Present17 AND Part_Present18
						AND Part_Present19 AND Part_Present20 AND Part_Present21
						AND Part_Present22 AND Part_Present23 AND Part_Present24
						AND Part_Present25 AND Part_Present26 AND Part_Present27
						AND Part_Present28 AND Part_Present29 AND Part_Present30
						AND Part_Present31 AND Part_Present32 AND Part_Present33
						AND Part_Present34 AND Part_Present35 AND Part_Present36
						AND Part_Present37 AND Part_Present38 AND Part_Present39
						AND Part_Present40)

					OR ((Model_ID=2)
						AND Part_Present1 AND Part_Present2 AND Part_Present3
						AND Part_Present4 AND Part_Present5 AND Part_Present6
						AND Part_Present7 AND Part_Present8 AND Part_Present9
						AND Part_Present10 AND Part_Present11 AND Part_Present12
						AND Part_Present13 AND Part_Present14 AND Part_Present15
						AND Part_Present16 AND Part_Present17 AND Part_Present18
						AND Part_Present19 AND Part_Present20 AND Part_Present21
						AND Part_Present22 AND Part_Present23 AND Part_Present24
						AND Part_Present25 AND Part_Present26 AND Part_Present27
						AND Part_Present28 AND Part_Present29 AND Part_Present30
						AND Part_Present31 AND Part_Present32 AND Part_Present33
						AND Part_Present34 AND Part_Present35 AND Part_Present36
						AND Part_Present37 AND Part_Present38 AND Part_Present39
						AND Part_Present40)

					OR ((Model_ID=3)
						AND Part_Present1 AND Part_Present2 AND Part_Present3
						AND Part_Present4 AND Part_Present5 AND Part_Present6
						AND Part_Present7 AND Part_Present8 AND Part_Present9
						AND Part_Present10 AND Part_Present11 AND Part_Present12
						AND Part_Present13 AND Part_Present14 AND Part_Present15
						AND Part_Present16 AND Part_Present17 AND Part_Present18
						AND Part_Present19 AND Part_Present20 AND Part_Present21
						AND Part_Present22 AND Part_Present23 AND Part_Present24
						AND Part_Present25 AND Part_Present26 AND Part_Present27
						AND Part_Present28 AND Part_Present29 AND Part_Present30
						AND Part_Present31 AND Part_Present32 AND Part_Present33
						AND Part_Present34 AND Part_Present35 AND Part_Present36
						AND Part_Present37 AND Part_Present38 AND Part_Present39
						AND Part_Present40)

					OR ((Model_ID=4)
						AND Part_Present1 AND Part_Present2 AND Part_Present3
						AND Part_Present4 AND Part_Present5 AND Part_Present6
						AND Part_Present7 AND Part_Present8 AND Part_Present9
						AND Part_Present10 AND Part_Present11 AND Part_Present12
						AND Part_Present13 AND Part_Present14 AND Part_Present15
						AND Part_Present16 AND Part_Present17 AND Part_Present18
						AND Part_Present19 AND Part_Present20 AND Part_Present21
						AND Part_Present22 AND Part_Present23 AND Part_Present24
						AND Part_Present25 AND Part_Present26 AND Part_Present27
						AND Part_Present28 AND Part_Present29 AND Part_Present30
						AND Part_Present31 AND Part_Present32 AND Part_Present33
						AND Part_Present34 AND Part_Present35 AND Part_Present36
						AND Part_Present37 AND Part_Present38 AND Part_Present39
						AND Part_Present40)
					) OR (All_Sensors_Off AND Dry_Cycle);


























(*end*)
END_ACTION

ACTION Cylinders:

(* -----------------------------------------------------------------------------------*)
(*Below are Examples only, each will have to be customized for your application
	Notes:
	- Use SODGxx-SSCC61x-xxxxxxx_Fix IO and Seq.xlsx document to capture Clamp / Cylinder I/O Layout
	- CLFaults1 thru 4 can be used to group cylinder type faults (All Clamps on CLFaults1, all Pins on CLFaults2)
		OR
	- CLFaults 1 thru 4 can be used to group cylinder UI screens 
		(All items on Cylinder_1.content screen are on CLFaults1, all items on Cylinder_2.content screen are on CLFaults2 as example)
*)
(* -----------------------------------------------------------------------------------*)



(*Clamps*)(*Clamps*)(*Clamps*)
(*Clamps*)(*Clamps*)(*Clamps*)
(*Clamps*)(*Clamps*)(*Clamps*)

		(*Clamp1*)
		Clamp1FB(
			Retracted_Sensor:= N02.I.0 ,
			Advanced_Sensor:= N02.I.1 ,
			Retract_Solenoid:= N100.Q.1,
			Advance_Solenoid:= N100.Q.0 ,
			Ret_Delay:= T#0.1S,
			Adv_Delay:= T#0.1S,
			Fault_Delay:= T#3.0S,
			Disable_Fault:= FALSE,
			In_Retracted_Position=> Clamp1RETD,
			In_Advanced_Position=> Clamp1ADVD,
			Faulted=> CLFaults1.1 );

		(*Clamp2*)
		Clamp2FB(
			Retracted_Sensor:= N02.I.2 ,
			Advanced_Sensor:= N02.I.3 ,
			Retract_Solenoid:= N100.Q.1 ,
			Advance_Solenoid:= N100.Q.0 ,
			Ret_Delay:= T#0.1S,
			Adv_Delay:= T#0.1S,
			Fault_Delay:= T#3.0S,
			Disable_Fault:= FALSE,
			In_Retracted_Position=> Clamp2RETD,
			In_Advanced_Position=> Clamp2ADVD,
			Faulted=> CLFaults1.2 );

		(*Clamp3*)
		Clamp3FB(
			Retracted_Sensor:= N02.I.4,
			Advanced_Sensor:= N02.I.5,
			Retract_Solenoid:= N100.Q.1,
			Advance_Solenoid:= N100.Q.0,
			Ret_Delay:= T#0.1S,
			Adv_Delay:= T#0.1S,
			Fault_Delay:= T#3.0S,
			Disable_Fault:= FALSE,
			In_Retracted_Position=> Clamp3RETD,
			In_Advanced_Position=> Clamp3ADVD,
			Faulted=> CLFaults1.3 );

		(*Clamp4*)
		Clamp4FB(
			Retracted_Sensor:= N02.I.6,
			Advanced_Sensor:= N02.I.7,
			Retract_Solenoid:= N100.Q.1,
			Advance_Solenoid:= N100.Q.0,
			Ret_Delay:= T#0.1S,
			Adv_Delay:= T#0.1S,
			Fault_Delay:= T#3.0S,
			Disable_Fault:= FALSE,
			In_Retracted_Position=> Clamp4RETD,
			In_Advanced_Position=> Clamp4ADVD,
			Faulted=> CLFaults1.4 );

		(*Clamp5*)
		Clamp5FB(
			Retracted_Sensor:= N03.I.0,
			Advanced_Sensor:= N03.I.1,
			Retract_Solenoid:= N100.Q.1,
			Advance_Solenoid:= N100.Q.0,
			Ret_Delay:= T#0.1S,
			Adv_Delay:= T#0.1S,
			Fault_Delay:= T#3.0S,
			Disable_Fault:= FALSE,
			In_Retracted_Position=> Clamp5RETD,
			In_Advanced_Position=> Clamp5ADVD,
			Faulted=> CLFaults1.5 );

		(*Clamp6*)
		Clamp6FB(
			Retracted_Sensor:= N03.I.2,
			Advanced_Sensor:= N03.I.3,
			Retract_Solenoid:= N100.Q.1,
			Advance_Solenoid:= N100.Q.0,
			Ret_Delay:= T#0.1S,
			Adv_Delay:= T#0.1S,
			Fault_Delay:= T#3.0S,
			Disable_Fault:= FALSE,
			In_Retracted_Position=> Clamp6RETD,
			In_Advanced_Position=> Clamp6ADVD,
			Faulted=> CLFaults1.6 );

		(*Clamp7*)
		Clamp7FB(
			Retracted_Sensor:= N03.I.4,
			Advanced_Sensor:= N03.I.5,
			Retract_Solenoid:= N100.Q.1,
			Advance_Solenoid:= N100.Q.0,
			Ret_Delay:= T#0.1S,
			Adv_Delay:= T#0.1S,
			Fault_Delay:= T#3.0S,
			Disable_Fault:= FALSE,
			In_Retracted_Position=> Clamp7RETD,
			In_Advanced_Position=> Clamp7ADVD,
			Faulted=> CLFaults1.7 );

		(*Clamp8*)
		Clamp8FB(
			Retracted_Sensor:= N03.I.6,
			Advanced_Sensor:= N03.I.7,
			Retract_Solenoid:= N100.Q.1,
			Advance_Solenoid:= N100.Q.0,
			Ret_Delay:= T#0.1S,
			Adv_Delay:= T#0.1S,
			Fault_Delay:= T#3.0S,
			Disable_Fault:= FALSE,
			In_Retracted_Position=> Clamp8RETD,
			In_Advanced_Position=> Clamp8ADVD,
			Faulted=> CLFaults1.8 );

		(*Clamp9*)
		Clamp9FB(
			Retracted_Sensor:= N04.I.0,
			Advanced_Sensor:= N04.I.1,
			Retract_Solenoid:= N100.Q.3,
			Advance_Solenoid:= N100.Q.2,
			Ret_Delay:= T#0.1S,
			Adv_Delay:= T#0.1S,
			Fault_Delay:= T#3.0S,
			Disable_Fault:= FALSE,
			In_Retracted_Position=> Clamp9RETD,
			In_Advanced_Position=> Clamp9ADVD,
			Faulted=> CLFaults1.9 );

		(*Clamp10*)
		Clamp10FB(
			Retracted_Sensor:= N04.I.2,
			Advanced_Sensor:= N04.I.3,
			Retract_Solenoid:= N100.Q.3,
			Advance_Solenoid:= N100.Q.2,
			Ret_Delay:= T#0.1S,
			Adv_Delay:= T#0.1S,
			Fault_Delay:= T#3.0S,
			Disable_Fault:= FALSE,
			In_Retracted_Position=> Clamp10RETD,
			In_Advanced_Position=> Clamp10ADVD,
			Faulted=> CLFaults1.10 );

		(*Clamp11*)
		Clamp11FB(
			Retracted_Sensor:= N04.I.4,
			Advanced_Sensor:= N04.I.5,
			Retract_Solenoid:= N100.Q.3,
			Advance_Solenoid:= N100.Q.2,
			Ret_Delay:= T#0.1S,
			Adv_Delay:= T#0.1S,
			Fault_Delay:= T#3.0S,
			Disable_Fault:= FALSE,
			In_Retracted_Position=> Clamp11RETD,
			In_Advanced_Position=> Clamp11ADVD,
			Faulted=> CLFaults1.11 );

		(*Clamp12*)
		Clamp12FB(
			Retracted_Sensor:= N04.I.6,
			Advanced_Sensor:= N04.I.7,
			Retract_Solenoid:= N100.Q.3,
			Advance_Solenoid:= N100.Q.2,
			Ret_Delay:= T#0.1S,
			Adv_Delay:= T#0.1S,
			Fault_Delay:= T#3.0S,
			Disable_Fault:= FALSE,
			In_Retracted_Position=> Clamp12RETD,
			In_Advanced_Position=> Clamp12ADVD,
			Faulted=> CLFaults1.12 );

		(*Clamp13*)
		Clamp13FB(
			Retracted_Sensor:= N05.I.0,
			Advanced_Sensor:= N05.I.1,
			Retract_Solenoid:= N100.Q.5,
			Advance_Solenoid:= N100.Q.4,
			Ret_Delay:= T#0.1S,
			Adv_Delay:= T#0.1S,
			Fault_Delay:= T#3.0S,
			Disable_Fault:= FALSE,
			In_Retracted_Position=> Clamp13RETD,
			In_Advanced_Position=> Clamp13ADVD,
			Faulted=> CLFaults1.13 );

		(*Clamp14*)
		Clamp14FB(
			Retracted_Sensor:= N05.I.2,
			Advanced_Sensor:= N05.I.3,
			Retract_Solenoid:= N100.Q.5,
			Advance_Solenoid:= N100.Q.4,
			Ret_Delay:= T#0.1S,
			Adv_Delay:= T#0.1S,
			Fault_Delay:= T#3.0S,
			Disable_Fault:= FALSE,
			In_Retracted_Position=> Clamp14RETD,
			In_Advanced_Position=> Clamp14ADVD,
			Faulted=> CLFaults1.14 );

		(*Clamp15*)
		Clamp15FB(
			Retracted_Sensor:= N05.I.4,
			Advanced_Sensor:= N05.I.5,
			Retract_Solenoid:= N100.Q.5,
			Advance_Solenoid:= N100.Q.4,
			Ret_Delay:= T#0.1S,
			Adv_Delay:= T#0.1S,
			Fault_Delay:= T#3.0S,
			Disable_Fault:= FALSE,
			In_Retracted_Position=> Clamp15RETD,
			In_Advanced_Position=> Clamp15ADVD,
			Faulted=> CLFaults1.15 );

		(*Clamp16*)
		Clamp16FB(
			Retracted_Sensor:= N05.I.6,
			Advanced_Sensor:= N05.I.7,
			Retract_Solenoid:= N100.Q.5,
			Advance_Solenoid:= N100.Q.4,
			Ret_Delay:= T#0.1S,
			Adv_Delay:= T#0.1S,
			Fault_Delay:= T#3.0S,
			Disable_Fault:= FALSE,
			In_Retracted_Position=> Clamp16RETD,
			In_Advanced_Position=> Clamp16ADVD,
			Faulted=> CLFaults1.16 );

		(*Clamp17*)
		Clamp17FB(
			Retracted_Sensor:= N06.I.0,
			Advanced_Sensor:= N06.I.1,
			Retract_Solenoid:= N100.Q.7,
			Advance_Solenoid:= N100.Q.6,
			Ret_Delay:= T#0.1S,
			Adv_Delay:= T#0.1S,
			Fault_Delay:= T#3.0S,
			Disable_Fault:= FALSE,
			In_Retracted_Position=> Clamp17RETD,
			In_Advanced_Position=> Clamp17ADVD,
			Faulted=> CLFaults1.17 );

		(*Clamp18*)
		Clamp18FB(
			Retracted_Sensor:= N06.I.2,
			Advanced_Sensor:= N06.I.3,
			Retract_Solenoid:= N100.Q.7,
			Advance_Solenoid:= N100.Q.6,
			Ret_Delay:= T#0.1S,
			Adv_Delay:= T#0.1S,
			Fault_Delay:= T#3.0S,
			Disable_Fault:= FALSE,
			In_Retracted_Position=> Clamp18RETD,
			In_Advanced_Position=> Clamp18ADVD,
			Faulted=> CLFaults1.18 );

		(*Clamp19*)
		Clamp19FB(
			Retracted_Sensor:= N06.I.4,
			Advanced_Sensor:= N06.I.5,
			Retract_Solenoid:= N100.Q.7,
			Advance_Solenoid:= N100.Q.6,
			Ret_Delay:= T#0.1S,
			Adv_Delay:= T#0.1S,
			Fault_Delay:= T#3.0S,
			Disable_Fault:= FALSE,
			In_Retracted_Position=> Clamp19RETD,
			In_Advanced_Position=> Clamp19ADVD,
			Faulted=> CLFaults1.19 );

		(*Clamp20*)
		Clamp20FB(
			Retracted_Sensor:= N06.I.6,
			Advanced_Sensor:= N06.I.7,
			Retract_Solenoid:= N100.Q.7,
			Advance_Solenoid:= N100.Q.6,
			Ret_Delay:= T#0.1S,
			Adv_Delay:= T#0.1S,
			Fault_Delay:= T#3.0S,
			Disable_Fault:= FALSE,
			In_Retracted_Position=> Clamp20RETD,
			In_Advanced_Position=> Clamp20ADVD,
			Faulted=> CLFaults1.20 );

		(*Clamp21*)
		Clamp21FB(
			Retracted_Sensor:= N07.I.0,
			Advanced_Sensor:= N07.I.1,
			Retract_Solenoid:= N100.Q.9,
			Advance_Solenoid:= N100.Q.8,
			Ret_Delay:= T#0.1S,
			Adv_Delay:= T#0.1S,
			Fault_Delay:= T#3.0S,
			Disable_Fault:= FALSE,
			In_Retracted_Position=> Clamp21RETD,
			In_Advanced_Position=> Clamp21ADVD,
			Faulted=> CLFaults1.21 );

		(*Clamp22*)
		Clamp22FB(
			Retracted_Sensor:= N07.I.2,
			Advanced_Sensor:= N07.I.3,
			Retract_Solenoid:= N100.Q.9,
			Advance_Solenoid:= N100.Q.8,
			Ret_Delay:= T#0.1S,
			Adv_Delay:= T#0.1S,
			Fault_Delay:= T#3.0S,
			Disable_Fault:= FALSE,
			In_Retracted_Position=> Clamp22RETD,
			In_Advanced_Position=> Clamp22ADVD,
			Faulted=> CLFaults1.22 );

		(*Clamp23*)
		Clamp23FB(
			Retracted_Sensor:= N07.I.4,
			Advanced_Sensor:= N07.I.5,
			Retract_Solenoid:= N100.Q.9,
			Advance_Solenoid:= N100.Q.8,
			Ret_Delay:= T#0.1S,
			Adv_Delay:= T#0.1S,
			Fault_Delay:= T#3.0S,
			Disable_Fault:= FALSE,
			In_Retracted_Position=> Clamp23RETD,
			In_Advanced_Position=> Clamp23ADVD,
			Faulted=> CLFaults1.23 );

		(*Clamp24*)
		Clamp24FB(
			Retracted_Sensor:= N07.I.6,
			Advanced_Sensor:= N07.I.7,
			Retract_Solenoid:= N100.Q.9,
			Advance_Solenoid:= N100.Q.8,
			Ret_Delay:= T#0.1S,
			Adv_Delay:= T#0.1S,
			Fault_Delay:= T#3.0S,
			Disable_Fault:= FALSE,
			In_Retracted_Position=> Clamp24RETD,
			In_Advanced_Position=> Clamp24ADVD,
			Faulted=> CLFaults1.24 );


(*Pins*)(*Pins*)(*Pins*)
(*Pins*)(*Pins*)(*Pins*)
(*Pins*)(*Pins*)(*Pins*)

		(*Pin1*)
		Pin1FB(
			Retracted_Sensor:= N03.I.0,
			Advanced_Sensor:= N03.I.1,
			Retract_Solenoid:= N101.Q.1,
			Advance_Solenoid:= N101.Q.0,
			Ret_Delay:= T#0.1S,
			Adv_Delay:= T#0.1S,
			Fault_Delay:= T#3.0S,
			Disable_Fault:= FALSE,
			In_Retracted_Position=> Pin1RETD,
			In_Advanced_Position=> Pin1ADVD,
			Faulted=> CLFaults2.1 );

		(*Pin2*)
		Pin2FB(
			Retracted_Sensor:= N03.I.2,
			Advanced_Sensor:= N03.I.3,
			Retract_Solenoid:= N101.Q.1,
			Advance_Solenoid:= N101.Q.0,
			Ret_Delay:= T#0.1S,
			Adv_Delay:= T#0.1S,
			Fault_Delay:= T#3.0S,
			Disable_Fault:= FALSE,
			In_Retracted_Position=> Pin2RETD,
			In_Advanced_Position=> Pin2ADVD,
			Faulted=> CLFaults2.2 );

		(*Pin3*)
		Pin3FB(
			Retracted_Sensor:= N03.I.4,
			Advanced_Sensor:= N03.I.5,
			Retract_Solenoid:= N101.Q.1,
			Advance_Solenoid:= N101.Q.0,
			Ret_Delay:= T#0.1S,
			Adv_Delay:= T#0.1S,
			Fault_Delay:= T#3.0S,
			Disable_Fault:= FALSE,
			In_Retracted_Position=> Pin3RETD,
			In_Advanced_Position=> Pin3ADVD,
			Faulted=> CLFaults2.3 );

